SPLINE
SPL {X  -159.245, Y  +707.432, Z    +0.000, E1   -21.244, E3 +348737.690}
SPL {X  -162.277, Y  +686.791, Z    +0.000, E1   -10.607, E3 +348739.101}
SPL {X  -162.766, Y  +677.687, Z    +0.000, E1    -5.239, E3 +348741.291}
SPL {X  -162.820, Y  +671.059, Z    +0.000, E1    -0.934, E3 +348741.647}
SPL {X  -162.820, Y  +666.960, Z    +0.000, E1    +2.343, E3 +348741.923}
SPL {X  -162.820, Y  +662.610, Z    +0.000, E1    +6.209, E3 +348741.950}
SPL {X  -162.820, Y  +654.280, Z    +0.000, E1   +14.617, E3 +348742.282}
SPL {X  -162.820, Y  +638.947, Z    +0.000, E1   +31.033, E3 +348740.336}
SPL {X  -162.820, Y  +608.150, Z    +0.000, E1   +43.921, E3 +348766.569}
SPL {X  -162.820, Y  +574.255, Z    +0.000, E1   +46.562, E3 +348816.362}
ENDSPLINE

SPLINE
SPL {X  -162.820, Y  +579.440, Z    +0.000, E1   +42.450, E3 +348829.550}
ENDSPLINE

SPLINE
SPL {X  -162.820, Y  +573.350, Z    +0.000, E1   +42.340, E3 +348844.228}
SPL {X  -162.820, Y  +565.899, Z    +0.000, E1   +42.413, E3 +348860.811}
SPL {X  -162.820, Y  +560.278, Z    +0.000, E1   +42.308, E3 +348874.149}
SPL {X  -162.820, Y  +555.861, Z    +0.000, E1   +42.349, E3 +348883.997}
SPL {X  -162.820, Y  +550.633, Z    +0.000, E1   +42.421, E3 +348895.527}
SPL {X  -162.820, Y  +546.534, Z    +0.000, E1   +42.268, E3 +348905.736}
SPL {X  -162.820, Y  +539.632, Z    +0.000, E1   +42.488, E3 +348920.458}
SPL {X  -162.820, Y  +533.959, Z    +0.000, E1   +42.310, E3 +348934.154}
SPL {X  -162.820, Y  +527.661, Z    +0.000, E1   +42.425, E3 +348948.150}
SPL {X  -162.820, Y  +521.246, Z    +0.000, E1   +42.365, E3 +348962.903}
SPL {X  -162.820, Y  +515.708, Z    +0.000, E1   +42.333, E3 +348975.865}
SPL {X  -162.820, Y  +508.859, Z    +0.000, E1   +42.416, E3 +348991.007}
SPL {X  -162.820, Y  +501.651, Z    +0.000, E1   +42.423, E3 +349007.483}
SPL {X  -162.820, Y  +494.841, Z    +0.000, E1   +42.316, E3 +349023.593}
SPL {X  -162.820, Y  +489.758, Z    +0.000, E1   +42.464, E3 +349034.186}
SPL {X  -162.820, Y  +485.695, Z    +0.000, E1   +42.386, E3 +349044.022}
SPL {X  -162.820, Y  +464.528, Z    +0.000, E1   +47.611, E3 +349057.099}
SPL {X  -162.820, Y  +459.899, Z    +0.000, E1   +47.097, E3 +349068.942}
SPL {X  -162.820, Y  +455.990, Z    +0.000, E1   +46.212, E3 +349082.016}
SPL {X  -162.820, Y  +452.032, Z    +0.000, E1   +45.224, E3 +349095.801}
SPL {X  -162.820, Y  +446.617, Z    +0.000, E1   +44.768, E3 +349109.888}
SPL {X  -162.820, Y  +437.902, Z    +0.000, E1   +44.900, E3 +349127.464}
SPL {X  -162.820, Y  +429.336, Z    +0.000, E1   +44.917, E3 +349145.231}
SPL {X  -162.820, Y  +423.193, Z    +0.000, E1   +44.819, E3 +349158.490}
SPL {X  -162.820, Y  +416.810, Z    +0.000, E1   +44.932, E3 +349171.378}
SPL {X  -162.820, Y  +408.782, Z    +0.000, E1   +44.820, E3 +349188.809}
SPL {X  -162.820, Y  +401.619, Z    +0.000, E1   +44.978, E3 +349202.731}
SPL {X  -162.820, Y  +394.771, Z    +0.000, E1   +44.856, E3 +349217.970}
SPL {X  -162.820, Y  +387.883, Z    +0.000, E1   +44.837, E3 +349232.324}
SPL {X  -162.820, Y  +382.755, Z    +0.000, E1   +44.828, E3 +349243.117}
SPL {X  -162.796, Y  +377.700, Z    +0.000, E1   +44.829, E3 +349253.697}
SPL {X  -162.619, Y  +372.412, Z    +0.000, E1   +44.928, E3 +349264.156}
SPL {X  -162.311, Y  +367.633, Z    +0.000, E1   +44.798, E3 +349274.923}
SPL {X  -161.766, Y  +362.002, Z    +0.000, E1   +44.644, E3 +349287.682}
SPL {X  -161.043, Y  +356.508, Z    +0.000, E1   +44.528, E3 +349299.797}
SPL {X  -160.417, Y  +352.631, Z    +0.000, E1   +44.411, E3 +349308.528}
SPL {X  -159.536, Y  +347.962, Z    +0.000, E1   +44.302, E3 +349319.054}
SPL {X  -158.195, Y  +341.969, Z    +0.000, E1   +44.082, E3 +349332.837}
SPL {X  -156.950, Y  +337.174, Z    +0.000, E1   +43.768, E3 +349344.527}
SPL {X  -155.654, Y  +332.729, Z    +0.000, E1   +43.534, E3 +349355.169}
SPL {X  -154.189, Y  +328.191, Z    +0.000, E1   +43.338, E3 +349365.666}
SPL {X  -149.333, Y  +315.614, Z    +0.000, E1   +46.650, E3 +349372.982}
SPL {X  -142.680, Y  +302.060, Z    +0.000, E1   +42.084, E3 +349439.326}
ENDSPLINE

SPLINE
SPL {X  -151.184, Y  +320.053, Z    +0.000, E1   +32.435, E3 +349506.569}
SPL {X  -158.917, Y  +345.064, Z    +0.000, E1   +21.858, E3 +349507.917}
SPL {X  -161.350, Y  +358.672, Z    +0.000, E1   +15.089, E3 +349510.620}
SPL {X  -162.491, Y  +370.147, Z    +0.000, E1    +8.815, E3 +349513.555}
SPL {X  -162.771, Y  +376.522, Z    +0.000, E1    +5.005, E3 +349513.164}
SPL {X  -162.820, Y  +381.116, Z    +0.000, E1    +2.017, E3 +349513.498}
SPL {X  -162.820, Y  +384.427, Z    +0.000, E1    -0.390, E3 +349513.902}
SPL {X  -162.820, Y  +387.736, Z    +0.000, E1    -3.142, E3 +349513.183}
SPL {X  -162.820, Y  +391.456, Z    +0.000, E1    -6.603, E3 +349513.969}
SPL {X  -162.820, Y  +397.032, Z    +0.000, E1   -12.435, E3 +349513.416}
SPL {X  -162.820, Y  +406.111, Z    +0.000, E1   -22.010, E3 +349514.468}
SPL {X  -162.820, Y  +418.653, Z    +0.000, E1   -36.657, E3 +349508.821}
SPL {X  -162.820, Y  +440.590, Z    +0.000, E1   -50.152, E3 +349514.066}
SPL {X  -162.820, Y  +447.889, Z    +0.000, E1   -43.424, E3 +349545.212}
SPL {X  -162.820, Y  +478.087, Z    +0.000, E1   -45.903, E3 +349590.431}
ENDSPLINE

SPLINE
SPL {X  -162.820, Y  +474.900, Z    +0.000, E1   -42.394, E3 +349604.583}
ENDSPLINE

SPLINE
SPL {X  -162.820, Y  +480.895, Z    +0.000, E1   -42.223, E3 +349619.245}
SPL {X  -162.820, Y  +485.782, Z    +0.000, E1   -42.348, E3 +349629.590}
SPL {X  -162.820, Y  +489.480, Z    +0.000, E1   -42.230, E3 +349638.818}
SPL {X  -162.820, Y  +494.825, Z    +0.000, E1   -42.287, E3 +349650.765}
SPL {X  -162.820, Y  +501.023, Z    +0.000, E1   -42.347, E3 +349664.647}
SPL {X  -162.820, Y  +506.968, Z    +0.000, E1   -42.248, E3 +349678.838}
SPL {X  -162.820, Y  +513.215, Z    +0.000, E1   -42.304, E3 +349692.812}
SPL {X  -162.820, Y  +518.708, Z    +0.000, E1   -42.272, E3 +349705.534}
SPL {X  -162.820, Y  +525.147, Z    +0.000, E1   -42.298, E3 +349720.276}
SPL {X  -162.820, Y  +531.715, Z    +0.000, E1   -42.312, E3 +349735.102}
SPL {X  -162.820, Y  +537.459, Z    +0.000, E1   -42.308, E3 +349748.361}
SPL {X  -162.820, Y  +542.643, Z    +0.000, E1   -42.173, E3 +349760.953}
SPL {X  -162.820, Y  +549.160, Z    +0.000, E1   -42.387, E3 +349774.712}
SPL {X  -162.820, Y  +554.884, Z    +0.000, E1   -42.207, E3 +349788.798}
SPL {X  -162.820, Y  +561.114, Z    +0.000, E1   -42.336, E3 +349802.378}
SPL {X  -162.820, Y  +566.097, Z    +0.000, E1   -42.118, E3 +349814.988}
SPL {X  -162.820, Y  +571.654, Z    +0.000, E1   -42.313, E3 +349826.641}
SPL {X  -162.820, Y  +577.246, Z    +0.000, E1   -42.284, E3 +349839.607}
SPL {X  -162.820, Y  +582.233, Z    +0.000, E1   -42.188, E3 +349851.586}
SPL {X  -162.820, Y  +588.138, Z    +0.000, E1   -42.308, E3 +349864.484}
SPL {X  -162.820, Y  +593.999, Z    +0.000, E1   -42.301, E3 +349877.894}
SPL {X  -162.820, Y  +599.194, Z    +0.000, E1   -42.235, E3 +349890.199}
SPL {X  -162.820, Y  +604.595, Z    +0.000, E1   -42.290, E3 +349902.230}
SPL {X  -162.820, Y  +609.630, Z    +0.000, E1   -42.276, E3 +349913.856}
SPL {X  -162.820, Y  +614.392, Z    +0.000, E1   -42.242, E3 +349924.956}
SPL {X  -162.820, Y  +618.928, Z    +0.000, E1   -42.220, E3 +349935.482}
SPL {X  -162.820, Y  +625.176, Z    +0.000, E1   -42.323, E3 +349949.334}
SPL {X  -162.820, Y  +631.865, Z    +0.000, E1   -42.327, E3 +349964.547}
SPL {X  -162.820, Y  +637.189, Z    +0.000, E1   -42.236, E3 +349977.221}
SPL {X  -162.820, Y  +642.066, Z    +0.000, E1   -42.247, E3 +349988.344}
SPL {X  -162.820, Y  +646.907, Z    +0.000, E1   -42.249, E3 +349999.463}
SPL {X  -162.820, Y  +652.374, Z    +0.000, E1   -42.262, E3 +350011.901}
SPL {X  -162.820, Y  +657.439, Z    +0.000, E1   -42.251, E3 +350023.574}
SPL {X  -162.820, Y  +663.328, Z    +0.000, E1   -42.283, E3 +350036.976}
SPL {X  -162.820, Y  +669.078, Z    +0.000, E1   -42.263, E3 +350050.172}
SPL {X  -162.819, Y  +673.910, Z    +0.000, E1   -42.244, E3 +350061.366}
SPL {X  -162.670, Y  +680.491, Z    +0.000, E1   -42.282, E3 +350076.409}
SPL {X  -162.151, Y  +688.243, Z    +0.000, E1   -42.207, E3 +350094.610}
SPL {X  -161.446, Y  +694.609, Z    +0.000, E1   -42.094, E3 +350109.692}
SPL {X  -160.889, Y  +698.503, Z    +0.000, E1   -41.849, E3 +350119.966}
SPL {X  -160.100, Y  +703.138, Z    +0.000, E1   -41.824, E3 +350130.824}
SPL {X  -158.994, Y  +708.588, Z    +0.000, E1   -41.616, E3 +350144.544}
SPL {X  -157.709, Y  +713.973, Z    +0.000, E1   -41.360, E3 +350158.326}
SPL {X  -156.530, Y  +718.319, Z    +0.000, E1   -41.164, E3 +350169.271}
SPL {X  -155.547, Y  +721.618, Z    +0.000, E1   -40.968, E3 +350177.894}
SPL {X  -151.388, Y  +733.433, Z    +0.000, E1   -44.269, E3 +350185.597}
SPL {X  -144.352, Y  +748.818, Z    +0.000, E1   -40.701, E3 +350254.632}
SPL {X  -143.859, Y  +749.757, Z    +0.000, E1   -39.148, E3 +350282.580}
ENDSPLINE

SPLINE
SPL {X  -159.245, Y  +707.432, Z    +0.000, E1   -21.244, E3 +350314.614}
SPL {X  -162.277, Y  +686.791, Z    +0.000, E1   -10.607, E3 +350316.024}
SPL {X  -162.766, Y  +677.687, Z    +0.000, E1    -5.239, E3 +350318.214}
SPL {X  -162.820, Y  +671.059, Z    +0.000, E1    -0.934, E3 +350318.570}
SPL {X  -162.820, Y  +666.960, Z    +0.000, E1    +2.343, E3 +350318.846}
SPL {X  -162.820, Y  +662.610, Z    +0.000, E1    +6.209, E3 +350318.873}
SPL {X  -162.820, Y  +654.280, Z    +0.000, E1   +14.617, E3 +350319.206}
SPL {X  -162.820, Y  +638.947, Z    +0.000, E1   +31.033, E3 +350317.259}
SPL {X  -162.820, Y  +608.150, Z    +0.000, E1   +43.921, E3 +350343.492}
SPL {X  -162.820, Y  +574.255, Z    +0.000, E1   +46.562, E3 +350393.286}
ENDSPLINE

SPLINE
SPL {X  -162.820, Y  +579.440, Z    +0.000, E1   +42.450, E3 +350406.473}
ENDSPLINE

SPLINE
SPL {X  -162.820, Y  +574.443, Z    +0.000, E1   +42.333, E3 +350418.568}
SPL {X  -162.820, Y  +568.554, Z    +0.000, E1   +42.362, E3 +350431.930}
SPL {X  -162.820, Y  +563.699, Z    +0.000, E1   +42.375, E3 +350442.787}
SPL {X  -162.820, Y  +560.278, Z    +0.000, E1   +42.308, E3 +350451.072}
SPL {X  -162.820, Y  +554.421, Z    +0.000, E1   +42.414, E3 +350463.940}
SPL {X  -162.820, Y  +547.774, Z    +0.000, E1   +42.344, E3 +350479.513}
SPL {X  -162.820, Y  +541.056, Z    +0.000, E1   +42.452, E3 +350494.175}
SPL {X  -162.820, Y  +535.223, Z    +0.000, E1   +42.386, E3 +350507.868}
SPL {X  -162.820, Y  +529.084, Z    +0.000, E1   +42.400, E3 +350521.791}
SPL {X  -162.820, Y  +522.568, Z    +0.000, E1   +42.385, E3 +350536.821}
SPL {X  -162.820, Y  +515.708, Z    +0.000, E1   +42.333, E3 +350552.788}
SPL {X  -162.820, Y  +510.265, Z    +0.000, E1   +42.390, E3 +350564.750}
SPL {X  -162.820, Y  +505.746, Z    +0.000, E1   +42.400, E3 +350575.063}
SPL {X  -162.820, Y  +500.461, Z    +0.000, E1   +42.387, E3 +350587.190}
SPL {X  -162.820, Y  +494.841, Z    +0.000, E1   +42.316, E3 +350600.516}
SPL {X  -162.820, Y  +487.903, Z    +0.000, E1   +42.488, E3 +350615.339}
SPL {X  -162.820, Y  +484.250, Z    +0.000, E1   +42.201, E3 +350625.200}
SPL {X  -162.820, Y  +464.528, Z    +0.000, E1   +47.611, E3 +350634.022}
SPL {X  -162.820, Y  +459.899, Z    +0.000, E1   +47.097, E3 +350645.865}
SPL {X  -162.820, Y  +455.990, Z    +0.000, E1   +46.212, E3 +350658.939}
SPL {X  -162.820, Y  +452.032, Z    +0.000, E1   +45.224, E3 +350672.724}
SPL {X  -162.820, Y  +446.617, Z    +0.000, E1   +44.768, E3 +350686.811}
SPL {X  -162.820, Y  +437.902, Z    +0.000, E1   +44.900, E3 +350704.388}
SPL {X  -162.820, Y  +430.894, Z    +0.000, E1   +44.976, E3 +350718.373}
SPL {X  -162.820, Y  +425.053, Z    +0.000, E1   +44.824, E3 +350731.635}
SPL {X  -162.820, Y  +418.403, Z    +0.000, E1   +44.941, E3 +350744.748}
SPL {X  -162.820, Y  +412.479, Z    +0.000, E1   +44.780, E3 +350758.179}
SPL {X  -162.820, Y  +406.707, Z    +0.000, E1   +44.849, E3 +350769.751}
SPL {X  -162.820, Y  +400.166, Z    +0.000, E1   +44.948, E3 +350783.036}
SPL {X  -162.820, Y  +393.279, Z    +0.000, E1   +44.825, E3 +350798.038}
SPL {X  -162.820, Y  +387.883, Z    +0.000, E1   +44.837, E3 +350809.247}
SPL {X  -162.820, Y  +382.755, Z    +0.000, E1   +44.828, E3 +350820.040}
SPL {X  -162.796, Y  +377.700, Z    +0.000, E1   +44.829, E3 +350830.620}
SPL {X  -162.619, Y  +372.412, Z    +0.000, E1   +44.928, E3 +350841.079}
SPL {X  -162.311, Y  +367.633, Z    +0.000, E1   +44.798, E3 +350851.846}
SPL {X  -161.766, Y  +362.002, Z    +0.000, E1   +44.644, E3 +350864.605}
SPL {X  -161.043, Y  +356.508, Z    +0.000, E1   +44.528, E3 +350876.720}
SPL {X  -160.070, Y  +350.699, Z    +0.000, E1   +44.409, E3 +350889.672}
SPL {X  -158.853, Y  +344.776, Z    +0.000, E1   +44.148, E3 +350903.492}
SPL {X  -157.292, Y  +338.433, Z    +0.000, E1   +43.917, E3 +350918.170}
SPL {X  -155.654, Y  +332.729, Z    +0.000, E1   +43.534, E3 +350932.092}
SPL {X  -154.189, Y  +328.191, Z    +0.000, E1   +43.338, E3 +350942.589}
SPL {X  -149.333, Y  +315.614, Z    +0.000, E1   +46.650, E3 +350949.905}
SPL {X  -142.680, Y  +302.060, Z    +0.000, E1   +42.084, E3 +351016.249}
ENDSPLINE

SPLINE
SPL {X  -151.184, Y  +320.053, Z    +0.000, E1   +32.435, E3 +351083.492}
SPL {X  -158.917, Y  +345.064, Z    +0.000, E1   +21.858, E3 +351084.840}
SPL {X  -161.350, Y  +358.672, Z    +0.000, E1   +15.089, E3 +351087.543}
SPL {X  -162.491, Y  +370.147, Z    +0.000, E1    +8.815, E3 +351090.478}
SPL {X  -162.771, Y  +376.522, Z    +0.000, E1    +5.005, E3 +351090.087}
SPL {X  -162.820, Y  +383.029, Z    +0.000, E1    +0.769, E3 +351090.655}
SPL {X  -162.820, Y  +387.736, Z    +0.000, E1    -3.142, E3 +351090.106}
SPL {X  -162.820, Y  +392.770, Z    +0.000, E1    -7.830, E3 +351090.758}
SPL {X  -162.820, Y  +398.469, Z    +0.000, E1   -14.078, E3 +351090.210}
SPL {X  -162.820, Y  +406.111, Z    +0.000, E1   -22.010, E3 +351091.391}
SPL {X  -162.820, Y  +418.653, Z    +0.000, E1   -36.657, E3 +351085.744}
SPL {X  -162.820, Y  +440.590, Z    +0.000, E1   -50.152, E3 +351090.989}
SPL {X  -162.820, Y  +447.889, Z    +0.000, E1   -43.424, E3 +351122.135}
SPL {X  -162.820, Y  +479.020, Z    +0.000, E1   -47.189, E3 +351161.711}
ENDSPLINE

SPLINE
SPL {X  -162.820, Y  +474.886, Z    +0.000, E1   -43.721, E3 +351173.596}
ENDSPLINE

SPLINE
SPL {X  -162.820, Y  +477.319, Z    +0.000, E1   -42.306, E3 +351187.521}
SPL {X  -162.820, Y  +483.923, Z    +0.000, E1   -42.291, E3 +351202.728}
SPL {X  -162.820, Y  +489.480, Z    +0.000, E1   -42.230, E3 +351215.741}
SPL {X  -162.820, Y  +494.825, Z    +0.000, E1   -42.287, E3 +351227.688}
SPL {X  -162.820, Y  +501.023, Z    +0.000, E1   -42.347, E3 +351241.570}
SPL {X  -162.820, Y  +506.968, Z    +0.000, E1   -42.248, E3 +351255.761}
SPL {X  -162.820, Y  +513.215, Z    +0.000, E1   -42.304, E3 +351269.735}
SPL {X  -162.820, Y  +518.708, Z    +0.000, E1   -42.272, E3 +351282.457}
SPL {X  -162.820, Y  +525.147, Z    +0.000, E1   -42.298, E3 +351297.199}
SPL {X  -162.820, Y  +531.715, Z    +0.000, E1   -42.312, E3 +351312.025}
SPL {X  -162.820, Y  +537.459, Z    +0.000, E1   -42.308, E3 +351325.284}
SPL {X  -162.820, Y  +542.643, Z    +0.000, E1   -42.173, E3 +351337.876}
SPL {X  -162.820, Y  +549.160, Z    +0.000, E1   -42.387, E3 +351351.635}
SPL {X  -162.820, Y  +554.884, Z    +0.000, E1   -42.207, E3 +351365.721}
SPL {X  -162.820, Y  +561.114, Z    +0.000, E1   -42.336, E3 +351379.301}
SPL {X  -162.820, Y  +566.097, Z    +0.000, E1   -42.118, E3 +351391.911}
SPL {X  -162.820, Y  +571.654, Z    +0.000, E1   -42.313, E3 +351403.564}
SPL {X  -162.820, Y  +577.246, Z    +0.000, E1   -42.284, E3 +351416.530}
SPL {X  -162.820, Y  +582.233, Z    +0.000, E1   -42.188, E3 +351428.509}
SPL {X  -162.820, Y  +588.138, Z    +0.000, E1   -42.308, E3 +351441.407}
SPL {X  -162.820, Y  +593.999, Z    +0.000, E1   -42.301, E3 +351454.817}
SPL {X  -162.820, Y  +599.194, Z    +0.000, E1   -42.235, E3 +351467.122}
SPL {X  -162.820, Y  +604.595, Z    +0.000, E1   -42.290, E3 +351479.153}
SPL {X  -162.820, Y  +609.630, Z    +0.000, E1   -42.276, E3 +351490.779}
SPL {X  -162.820, Y  +614.392, Z    +0.000, E1   -42.242, E3 +351501.879}
SPL {X  -162.820, Y  +620.424, Z    +0.000, E1   -42.277, E3 +351515.627}
SPL {X  -162.820, Y  +626.430, Z    +0.000, E1   -42.291, E3 +351529.177}
SPL {X  -162.820, Y  +631.865, Z    +0.000, E1   -42.327, E3 +351541.470}
SPL {X  -162.820, Y  +637.189, Z    +0.000, E1   -42.236, E3 +351554.144}
SPL {X  -162.820, Y  +642.066, Z    +0.000, E1   -42.247, E3 +351565.267}
SPL {X  -162.820, Y  +646.907, Z    +0.000, E1   -42.249, E3 +351576.386}
SPL {X  -162.820, Y  +652.374, Z    +0.000, E1   -42.262, E3 +351588.824}
SPL {X  -162.820, Y  +657.439, Z    +0.000, E1   -42.251, E3 +351600.497}
SPL {X  -162.820, Y  +663.328, Z    +0.000, E1   -42.283, E3 +351613.899}
SPL {X  -162.820, Y  +669.078, Z    +0.000, E1   -42.263, E3 +351627.095}
SPL {X  -162.819, Y  +673.910, Z    +0.000, E1   -42.244, E3 +351638.289}
SPL {X  -162.729, Y  +678.944, Z    +0.000, E1   -42.273, E3 +351649.657}
SPL {X  -162.479, Y  +684.035, Z    +0.000, E1   -42.168, E3 +351661.994}
SPL {X  -162.026, Y  +689.560, Z    +0.000, E1   -42.192, E3 +351674.483}
SPL {X  -161.446, Y  +694.609, Z    +0.000, E1   -42.094, E3 +351686.615}
SPL {X  -160.681, Y  +699.806, Z    +0.000, E1   -41.866, E3 +351699.898}
SPL {X  -159.658, Y  +705.434, Z    +0.000, E1   -41.735, E3 +351713.528}
SPL {X  -158.727, Y  +709.780, Z    +0.000, E1   -41.560, E3 +351724.395}
SPL {X  -157.709, Y  +713.973, Z    +0.000, E1   -41.360, E3 +351735.249}
SPL {X  -156.530, Y  +718.319, Z    +0.000, E1   -41.164, E3 +351746.194}
SPL {X  -155.547, Y  +721.618, Z    +0.000, E1   -40.968, E3 +351754.818}
SPL {X  -151.388, Y  +733.433, Z    +0.000, E1   -44.269, E3 +351762.520}
SPL {X  -144.352, Y  +748.818, Z    +0.000, E1   -40.701, E3 +351831.555}
SPL {X  -143.859, Y  +749.757, Z    +0.000, E1   -39.148, E3 +351859.503}
ENDSPLINE

SPLINE
SPL {X  -159.245, Y  +707.432, Z    +0.000, E1   -21.244, E3 +351891.537}
SPL {X  -162.277, Y  +686.791, Z    +0.000, E1   -10.607, E3 +351892.947}
SPL {X  -162.766, Y  +677.687, Z    +0.000, E1    -5.239, E3 +351895.137}
SPL {X  -162.820, Y  +672.396, Z    +0.000, E1    -1.801, E3 +351895.925}
SPL {X  -162.820, Y  +667.851, Z    +0.000, E1    +1.551, E3 +351895.422}
SPL {X  -162.820, Y  +664.036, Z    +0.000, E1    +4.934, E3 +351896.141}
SPL {X  -162.820, Y  +661.024, Z    +0.000, E1    +7.880, E3 +351895.411}
SPL {X  -162.820, Y  +656.051, Z    +0.000, E1   +12.848, E3 +351896.278}
SPL {X  -162.820, Y  +650.794, Z    +0.000, E1   +18.580, E3 +351895.834}
SPL {X  -162.820, Y  +638.947, Z    +0.000, E1   +31.033, E3 +351894.182}
SPL {X  -162.820, Y  +608.150, Z    +0.000, E1   +43.921, E3 +351920.415}
SPL {X  -162.820, Y  +574.255, Z    +0.000, E1   +46.562, E3 +351970.209}
ENDSPLINE

SPLINE
SPL {X  -162.820, Y  +579.440, Z    +0.000, E1   +42.450, E3 +351983.396}
ENDSPLINE

SPLINE
SPL {X  -162.820, Y  +573.350, Z    +0.000, E1   +42.340, E3 +351998.074}
SPL {X  -162.820, Y  +565.899, Z    +0.000, E1   +42.413, E3 +352014.657}
SPL {X  -162.820, Y  +560.278, Z    +0.000, E1   +42.308, E3 +352027.995}
SPL {X  -162.820, Y  +554.421, Z    +0.000, E1   +42.414, E3 +352040.863}
SPL {X  -162.820, Y  +547.774, Z    +0.000, E1   +42.344, E3 +352056.436}
SPL {X  -162.820, Y  +541.056, Z    +0.000, E1   +42.452, E3 +352071.098}
SPL {X  -162.820, Y  +535.223, Z    +0.000, E1   +42.386, E3 +352084.791}
SPL {X  -162.820, Y  +529.084, Z    +0.000, E1   +42.400, E3 +352098.714}
SPL {X  -162.820, Y  +524.911, Z    +0.000, E1   +42.325, E3 +352108.560}
SPL {X  -162.820, Y  +519.984, Z    +0.000, E1   +42.385, E3 +352119.631}
SPL {X  -162.820, Y  +514.684, Z    +0.000, E1   +42.289, E3 +352132.202}
SPL {X  -162.820, Y  +508.859, Z    +0.000, E1   +42.416, E3 +352144.853}
SPL {X  -162.820, Y  +501.651, Z    +0.000, E1   +42.423, E3 +352161.329}
SPL {X  -162.820, Y  +496.578, Z    +0.000, E1   +42.329, E3 +352173.237}
SPL {X  -162.820, Y  +491.918, Z    +0.000, E1   +42.382, E3 +352183.731}
SPL {X  -162.820, Y  +485.695, Z    +0.000, E1   +42.386, E3 +352197.868}
SPL {X  -162.820, Y  +464.528, Z    +0.000, E1   +47.611, E3 +352210.946}
SPL {X  -162.820, Y  +459.899, Z    +0.000, E1   +47.097, E3 +352222.788}
SPL {X  -162.820, Y  +455.990, Z    +0.000, E1   +46.212, E3 +352235.862}
SPL {X  -162.820, Y  +452.032, Z    +0.000, E1   +45.224, E3 +352249.647}
SPL {X  -162.820, Y  +446.617, Z    +0.000, E1   +44.768, E3 +352263.734}
SPL {X  -162.820, Y  +437.902, Z    +0.000, E1   +44.900, E3 +352281.311}
SPL {X  -162.820, Y  +430.894, Z    +0.000, E1   +44.976, E3 +352295.296}
SPL {X  -162.820, Y  +425.053, Z    +0.000, E1   +44.824, E3 +352308.558}
SPL {X  -162.820, Y  +418.403, Z    +0.000, E1   +44.941, E3 +352321.671}
SPL {X  -162.820, Y  +412.479, Z    +0.000, E1   +44.780, E3 +352335.102}
SPL {X  -162.820, Y  +406.707, Z    +0.000, E1   +44.849, E3 +352346.674}
SPL {X  -162.820, Y  +401.619, Z    +0.000, E1   +44.978, E3 +352356.577}
SPL {X  -162.820, Y  +394.771, Z    +0.000, E1   +44.856, E3 +352371.816}
SPL {X  -162.820, Y  +387.883, Z    +0.000, E1   +44.837, E3 +352386.170}
SPL {X  -162.820, Y  +382.755, Z    +0.000, E1   +44.828, E3 +352396.963}
SPL {X  -162.796, Y  +377.700, Z    +0.000, E1   +44.829, E3 +352407.543}
SPL {X  -162.619, Y  +372.412, Z    +0.000, E1   +44.928, E3 +352418.002}
SPL {X  -162.311, Y  +367.633, Z    +0.000, E1   +44.798, E3 +352428.769}
SPL {X  -161.766, Y  +362.002, Z    +0.000, E1   +44.644, E3 +352441.528}
SPL {X  -161.043, Y  +356.508, Z    +0.000, E1   +44.528, E3 +352453.643}
SPL {X  -160.417, Y  +352.631, Z    +0.000, E1   +44.411, E3 +352462.374}
SPL {X  -159.536, Y  +347.962, Z    +0.000, E1   +44.302, E3 +352472.900}
SPL {X  -158.195, Y  +341.969, Z    +0.000, E1   +44.082, E3 +352486.683}
SPL {X  -156.950, Y  +337.174, Z    +0.000, E1   +43.768, E3 +352498.374}
SPL {X  -155.654, Y  +332.729, Z    +0.000, E1   +43.534, E3 +352509.015}
SPL {X  -153.067, Y  +324.996, Z    +0.000, E1   +44.257, E3 +352521.069}
SPL {X  -147.786, Y  +312.164, Z    +0.000, E1   +47.292, E3 +352529.800}
SPL {X  -142.680, Y  +302.060, Z    +0.000, E1   +42.084, E3 +352593.172}
ENDSPLINE

SPLINE
SPL {X  -151.184, Y  +320.053, Z    +0.000, E1   +32.435, E3 +352660.415}
SPL {X  -158.917, Y  +345.064, Z    +0.000, E1   +21.858, E3 +352661.763}
SPL {X  -161.350, Y  +358.672, Z    +0.000, E1   +15.089, E3 +352664.466}
SPL {X  -162.491, Y  +370.147, Z    +0.000, E1    +8.815, E3 +352667.401}
SPL {X  -162.816, Y  +379.394, Z    +0.000, E1    +3.267, E3 +352667.229}
SPL {X  -162.820, Y  +384.427, Z    +0.000, E1    -0.390, E3 +352667.748}
SPL {X  -162.820, Y  +387.736, Z    +0.000, E1    -3.142, E3 +352667.029}
SPL {X  -162.820, Y  +392.770, Z    +0.000, E1    -7.830, E3 +352667.681}
SPL {X  -162.820, Y  +398.469, Z    +0.000, E1   -14.078, E3 +352667.134}
SPL {X  -162.820, Y  +406.111, Z    +0.000, E1   -22.010, E3 +352668.314}
SPL {X  -162.820, Y  +418.653, Z    +0.000, E1   -36.657, E3 +352662.667}
SPL {X  -162.820, Y  +440.590, Z    +0.000, E1   -50.152, E3 +352667.912}
SPL {X  -162.820, Y  +447.889, Z    +0.000, E1   -43.424, E3 +352699.058}
SPL {X  -162.820, Y  +479.020, Z    +0.000, E1   -47.189, E3 +352738.634}
ENDSPLINE

SPLINE
SPL {X  -162.820, Y  +474.886, Z    +0.000, E1   -43.721, E3 +352750.519}
ENDSPLINE

SPLINE
SPL {X  -162.820, Y  +477.319, Z    +0.000, E1   -42.306, E3 +352764.444}
SPL {X  -162.820, Y  +483.923, Z    +0.000, E1   -42.291, E3 +352779.651}
SPL {X  -162.820, Y  +489.480, Z    +0.000, E1   -42.230, E3 +352792.664}
SPL {X  -162.820, Y  +494.825, Z    +0.000, E1   -42.287, E3 +352804.611}
SPL {X  -162.820, Y  +501.023, Z    +0.000, E1   -42.347, E3 +352818.493}
SPL {X  -162.820, Y  +506.968, Z    +0.000, E1   -42.248, E3 +352832.684}
SPL {X  -162.820, Y  +513.215, Z    +0.000, E1   -42.304, E3 +352846.658}
SPL {X  -162.820, Y  +518.708, Z    +0.000, E1   -42.272, E3 +352859.380}
SPL {X  -162.820, Y  +525.147, Z    +0.000, E1   -42.298, E3 +352874.122}
SPL {X  -162.820, Y  +531.715, Z    +0.000, E1   -42.312, E3 +352888.948}
SPL {X  -162.820, Y  +537.459, Z    +0.000, E1   -42.308, E3 +352902.207}
SPL {X  -162.820, Y  +542.643, Z    +0.000, E1   -42.173, E3 +352914.799}
SPL {X  -162.820, Y  +549.160, Z    +0.000, E1   -42.387, E3 +352928.558}
SPL {X  -162.820, Y  +554.884, Z    +0.000, E1   -42.207, E3 +352942.644}
SPL {X  -162.820, Y  +561.114, Z    +0.000, E1   -42.336, E3 +352956.224}
SPL {X  -162.820, Y  +566.097, Z    +0.000, E1   -42.118, E3 +352968.834}
SPL {X  -162.820, Y  +571.654, Z    +0.000, E1   -42.313, E3 +352980.487}
SPL {X  -162.820, Y  +577.246, Z    +0.000, E1   -42.284, E3 +352993.453}
SPL {X  -162.820, Y  +582.233, Z    +0.000, E1   -42.188, E3 +353005.432}
SPL {X  -162.820, Y  +588.138, Z    +0.000, E1   -42.308, E3 +353018.330}
SPL {X  -162.820, Y  +593.999, Z    +0.000, E1   -42.301, E3 +353031.740}
SPL {X  -162.820, Y  +599.194, Z    +0.000, E1   -42.235, E3 +353044.045}
SPL {X  -162.820, Y  +604.595, Z    +0.000, E1   -42.290, E3 +353056.076}
SPL {X  -162.820, Y  +609.630, Z    +0.000, E1   -42.276, E3 +353067.702}
SPL {X  -162.820, Y  +614.392, Z    +0.000, E1   -42.242, E3 +353078.802}
SPL {X  -162.820, Y  +620.424, Z    +0.000, E1   -42.277, E3 +353092.550}
SPL {X  -162.820, Y  +626.430, Z    +0.000, E1   -42.291, E3 +353106.100}
SPL {X  -162.820, Y  +631.865, Z    +0.000, E1   -42.327, E3 +353118.393}
SPL {X  -162.820, Y  +637.189, Z    +0.000, E1   -42.236, E3 +353131.067}
SPL {X  -162.820, Y  +642.066, Z    +0.000, E1   -42.247, E3 +353142.190}
SPL {X  -162.820, Y  +646.907, Z    +0.000, E1   -42.249, E3 +353153.309}
SPL {X  -162.820, Y  +652.374, Z    +0.000, E1   -42.262, E3 +353165.747}
SPL {X  -162.820, Y  +658.634, Z    +0.000, E1   -42.281, E3 +353180.104}
SPL {X  -162.820, Y  +664.480, Z    +0.000, E1   -42.257, E3 +353193.499}
SPL {X  -162.820, Y  +669.078, Z    +0.000, E1   -42.263, E3 +353204.018}
SPL {X  -162.819, Y  +673.910, Z    +0.000, E1   -42.244, E3 +353215.212}
SPL {X  -162.729, Y  +678.944, Z    +0.000, E1   -42.273, E3 +353226.580}
SPL {X  -162.479, Y  +684.035, Z    +0.000, E1   -42.168, E3 +353238.917}
SPL {X  -162.026, Y  +689.560, Z    +0.000, E1   -42.192, E3 +353251.406}
SPL {X  -161.446, Y  +694.609, Z    +0.000, E1   -42.094, E3 +353263.538}
SPL {X  -160.681, Y  +699.806, Z    +0.000, E1   -41.866, E3 +353276.821}
SPL {X  -159.658, Y  +705.434, Z    +0.000, E1   -41.735, E3 +353290.451}
SPL {X  -158.502, Y  +710.748, Z    +0.000, E1   -41.532, E3 +353303.798}
SPL {X  -157.452, Y  +714.962, Z    +0.000, E1   -41.276, E3 +353314.794}
SPL {X  -156.530, Y  +718.319, Z    +0.000, E1   -41.164, E3 +353323.117}
SPL {X  -155.547, Y  +721.618, Z    +0.000, E1   -40.968, E3 +353331.741}
SPL {X  -151.388, Y  +733.433, Z    +0.000, E1   -44.269, E3 +353339.443}
SPL {X  -144.352, Y  +748.818, Z    +0.000, E1   -40.701, E3 +353408.478}
SPL {X  -143.859, Y  +749.757, Z    +0.000, E1   -39.148, E3 +353436.426}
ENDSPLINE

SPLINE
SPL {X  -159.245, Y  +707.432, Z    +0.000, E1   -21.244, E3 +353468.460}
SPL {X  -162.277, Y  +686.791, Z    +0.000, E1   -10.607, E3 +353469.870}
SPL {X  -162.766, Y  +677.687, Z    +0.000, E1    -5.239, E3 +353472.060}
SPL {X  -162.820, Y  +671.059, Z    +0.000, E1    -0.934, E3 +353472.416}
SPL {X  -162.820, Y  +666.960, Z    +0.000, E1    +2.343, E3 +353472.692}
SPL {X  -162.820, Y  +662.610, Z    +0.000, E1    +6.209, E3 +353472.719}
SPL {X  -162.820, Y  +654.280, Z    +0.000, E1   +14.617, E3 +353473.052}
SPL {X  -162.820, Y  +638.947, Z    +0.000, E1   +31.033, E3 +353471.105}
SPL {X  -162.820, Y  +608.150, Z    +0.000, E1   +43.921, E3 +353497.338}
SPL {X  -162.820, Y  +574.255, Z    +0.000, E1   +46.562, E3 +353547.132}
ENDSPLINE

SPLINE
SPL {X  -162.820, Y  +579.440, Z    +0.000, E1   +42.450, E3 +353560.319}
ENDSPLINE

SPLINE
SPL {X  -162.820, Y  +574.443, Z    +0.000, E1   +42.333, E3 +353572.414}
SPL {X  -162.820, Y  +568.554, Z    +0.000, E1   +42.362, E3 +353585.776}
SPL {X  -162.820, Y  +561.474, Z    +0.000, E1   +42.369, E3 +353601.961}
SPL {X  -162.820, Y  +554.421, Z    +0.000, E1   +42.414, E3 +353617.786}
SPL {X  -162.820, Y  +547.774, Z    +0.000, E1   +42.344, E3 +353633.359}
SPL {X  -162.820, Y  +541.056, Z    +0.000, E1   +42.452, E3 +353648.021}
SPL {X  -162.820, Y  +535.223, Z    +0.000, E1   +42.386, E3 +353661.714}
SPL {X  -162.820, Y  +529.084, Z    +0.000, E1   +42.400, E3 +353675.637}
SPL {X  -162.820, Y  +522.568, Z    +0.000, E1   +42.385, E3 +353690.667}
SPL {X  -162.820, Y  +515.708, Z    +0.000, E1   +42.333, E3 +353706.634}
SPL {X  -162.820, Y  +508.859, Z    +0.000, E1   +42.416, E3 +353721.776}
SPL {X  -162.820, Y  +501.651, Z    +0.000, E1   +42.423, E3 +353738.252}
SPL {X  -162.820, Y  +494.841, Z    +0.000, E1   +42.316, E3 +353754.362}
SPL {X  -162.820, Y  +486.958, Z    +0.000, E1   +42.460, E3 +353771.655}
SPL {X  -162.820, Y  +466.305, Z    +0.000, E1   +47.564, E3 +353784.662}
SPL {X  -162.820, Y  +460.790, Z    +0.000, E1   +47.323, E3 +353796.838}
SPL {X  -162.820, Y  +455.990, Z    +0.000, E1   +46.212, E3 +353812.785}
SPL {X  -162.820, Y  +452.032, Z    +0.000, E1   +45.224, E3 +353826.570}
SPL {X  -162.820, Y  +446.617, Z    +0.000, E1   +44.768, E3 +353840.657}
SPL {X  -162.820, Y  +437.902, Z    +0.000, E1   +44.900, E3 +353858.234}
SPL {X  -162.820, Y  +430.894, Z    +0.000, E1   +44.976, E3 +353872.219}
SPL {X  -162.820, Y  +425.053, Z    +0.000, E1   +44.824, E3 +353885.481}
SPL {X  -162.820, Y  +416.810, Z    +0.000, E1   +44.932, E3 +353902.148}
SPL {X  -162.820, Y  +408.782, Z    +0.000, E1   +44.820, E3 +353919.578}
SPL {X  -162.820, Y  +401.619, Z    +0.000, E1   +44.978, E3 +353933.500}
SPL {X  -162.820, Y  +394.771, Z    +0.000, E1   +44.856, E3 +353948.739}
SPL {X  -162.820, Y  +387.883, Z    +0.000, E1   +44.837, E3 +353963.093}
SPL {X  -162.820, Y  +382.755, Z    +0.000, E1   +44.828, E3 +353973.886}
SPL {X  -162.796, Y  +377.700, Z    +0.000, E1   +44.829, E3 +353984.466}
SPL {X  -162.619, Y  +372.412, Z    +0.000, E1   +44.928, E3 +353994.925}
SPL {X  -162.311, Y  +367.633, Z    +0.000, E1   +44.798, E3 +354005.693}
SPL {X  -161.766, Y  +362.002, Z    +0.000, E1   +44.644, E3 +354018.451}
SPL {X  -161.043, Y  +356.508, Z    +0.000, E1   +44.528, E3 +354030.566}
SPL {X  -160.070, Y  +350.699, Z    +0.000, E1   +44.409, E3 +354043.518}
SPL {X  -158.853, Y  +344.776, Z    +0.000, E1   +44.148, E3 +354057.338}
SPL {X  -157.292, Y  +338.433, Z    +0.000, E1   +43.917, E3 +354072.017}
SPL {X  -155.654, Y  +332.729, Z    +0.000, E1   +43.534, E3 +354085.938}
SPL {X  -154.189, Y  +328.191, Z    +0.000, E1   +43.338, E3 +354096.435}
SPL {X  -149.333, Y  +315.614, Z    +0.000, E1   +46.650, E3 +354103.751}
SPL {X  -142.680, Y  +302.060, Z    +0.000, E1   +42.084, E3 +354170.095}
ENDSPLINE

SPLINE
SPL {X  -151.184, Y  +320.053, Z    +0.000, E1   +32.435, E3 +354237.338}
SPL {X  -158.917, Y  +345.064, Z    +0.000, E1   +21.858, E3 +354238.687}
SPL {X  -161.350, Y  +358.672, Z    +0.000, E1   +15.089, E3 +354241.389}
SPL {X  -162.491, Y  +370.147, Z    +0.000, E1    +8.815, E3 +354244.324}
SPL {X  -162.771, Y  +376.522, Z    +0.000, E1    +5.005, E3 +354243.933}
SPL {X  -162.820, Y  +383.029, Z    +0.000, E1    +0.769, E3 +354244.501}
SPL {X  -162.820, Y  +387.736, Z    +0.000, E1    -3.142, E3 +354243.952}
SPL {X  -162.820, Y  +392.770, Z    +0.000, E1    -7.830, E3 +354244.604}
SPL {X  -162.820, Y  +398.469, Z    +0.000, E1   -14.078, E3 +354244.057}
SPL {X  -162.820, Y  +406.111, Z    +0.000, E1   -22.010, E3 +354245.237}
SPL {X  -162.820, Y  +418.653, Z    +0.000, E1   -36.657, E3 +354239.590}
SPL {X  -162.820, Y  +440.590, Z    +0.000, E1   -50.152, E3 +354244.835}
SPL {X  -162.820, Y  +447.889, Z    +0.000, E1   -43.424, E3 +354275.981}
SPL {X  -162.820, Y  +478.087, Z    +0.000, E1   -45.903, E3 +354321.200}
ENDSPLINE

SPLINE
SPL {X  -162.820, Y  +474.900, Z    +0.000, E1   -42.394, E3 +354335.353}
ENDSPLINE

SPLINE
SPL {X  -162.820, Y  +480.895, Z    +0.000, E1   -42.223, E3 +354350.014}
SPL {X  -162.820, Y  +485.782, Z    +0.000, E1   -42.348, E3 +354360.360}
SPL {X  -162.820, Y  +489.480, Z    +0.000, E1   -42.230, E3 +354369.587}
SPL {X  -162.820, Y  +494.825, Z    +0.000, E1   -42.287, E3 +354381.534}
SPL {X  -162.820, Y  +501.023, Z    +0.000, E1   -42.347, E3 +354395.416}
SPL {X  -162.820, Y  +506.968, Z    +0.000, E1   -42.248, E3 +354409.607}
SPL {X  -162.820, Y  +513.215, Z    +0.000, E1   -42.304, E3 +354423.582}
SPL {X  -162.820, Y  +518.708, Z    +0.000, E1   -42.272, E3 +354436.303}
SPL {X  -162.820, Y  +525.147, Z    +0.000, E1   -42.298, E3 +354451.045}
SPL {X  -162.820, Y  +531.715, Z    +0.000, E1   -42.312, E3 +354465.871}
SPL {X  -162.820, Y  +537.459, Z    +0.000, E1   -42.308, E3 +354479.130}
SPL {X  -162.820, Y  +542.643, Z    +0.000, E1   -42.173, E3 +354491.723}
SPL {X  -162.820, Y  +549.160, Z    +0.000, E1   -42.387, E3 +354505.481}
SPL {X  -162.820, Y  +554.884, Z    +0.000, E1   -42.207, E3 +354519.567}
SPL {X  -162.820, Y  +561.114, Z    +0.000, E1   -42.336, E3 +354533.147}
SPL {X  -162.820, Y  +566.097, Z    +0.000, E1   -42.118, E3 +354545.757}
SPL {X  -162.820, Y  +571.654, Z    +0.000, E1   -42.313, E3 +354557.410}
SPL {X  -162.820, Y  +577.246, Z    +0.000, E1   -42.284, E3 +354570.376}
SPL {X  -162.820, Y  +582.233, Z    +0.000, E1   -42.188, E3 +354582.355}
SPL {X  -162.820, Y  +588.138, Z    +0.000, E1   -42.308, E3 +354595.253}
SPL {X  -162.820, Y  +593.999, Z    +0.000, E1   -42.301, E3 +354608.663}
SPL {X  -162.820, Y  +599.194, Z    +0.000, E1   -42.235, E3 +354620.968}
SPL {X  -162.820, Y  +604.595, Z    +0.000, E1   -42.290, E3 +354633.000}
SPL {X  -162.820, Y  +609.630, Z    +0.000, E1   -42.276, E3 +354644.625}
SPL {X  -162.820, Y  +614.392, Z    +0.000, E1   -42.242, E3 +354655.726}
SPL {X  -162.820, Y  +620.424, Z    +0.000, E1   -42.277, E3 +354669.473}
SPL {X  -162.820, Y  +626.430, Z    +0.000, E1   -42.291, E3 +354683.023}
SPL {X  -162.820, Y  +631.865, Z    +0.000, E1   -42.327, E3 +354695.317}
SPL {X  -162.820, Y  +637.189, Z    +0.000, E1   -42.236, E3 +354707.991}
SPL {X  -162.820, Y  +642.066, Z    +0.000, E1   -42.247, E3 +354719.113}
SPL {X  -162.820, Y  +646.907, Z    +0.000, E1   -42.249, E3 +354730.232}
SPL {X  -162.820, Y  +652.374, Z    +0.000, E1   -42.262, E3 +354742.670}
SPL {X  -162.820, Y  +657.439, Z    +0.000, E1   -42.251, E3 +354754.343}
SPL {X  -162.820, Y  +663.328, Z    +0.000, E1   -42.283, E3 +354767.745}
SPL {X  -162.820, Y  +669.078, Z    +0.000, E1   -42.263, E3 +354780.941}
SPL {X  -162.819, Y  +673.910, Z    +0.000, E1   -42.244, E3 +354792.136}
SPL {X  -162.729, Y  +678.944, Z    +0.000, E1   -42.273, E3 +354803.503}
SPL {X  -162.479, Y  +684.035, Z    +0.000, E1   -42.168, E3 +354815.841}
SPL {X  -162.026, Y  +689.560, Z    +0.000, E1   -42.192, E3 +354828.329}
SPL {X  -161.446, Y  +694.609, Z    +0.000, E1   -42.094, E3 +354840.461}
SPL {X  -160.889, Y  +698.503, Z    +0.000, E1   -41.849, E3 +354850.735}
SPL {X  -160.100, Y  +703.138, Z    +0.000, E1   -41.824, E3 +354861.594}
SPL {X  -158.994, Y  +708.588, Z    +0.000, E1   -41.616, E3 +354875.313}
SPL {X  -157.709, Y  +713.973, Z    +0.000, E1   -41.360, E3 +354889.095}
SPL {X  -156.530, Y  +718.319, Z    +0.000, E1   -41.164, E3 +354900.040}
SPL {X  -155.547, Y  +721.618, Z    +0.000, E1   -40.968, E3 +354908.664}
SPL {X  -151.388, Y  +733.433, Z    +0.000, E1   -44.269, E3 +354916.366}
SPL {X  -144.352, Y  +748.818, Z    +0.000, E1   -40.701, E3 +354985.401}
SPL {X  -143.859, Y  +749.757, Z    +0.000, E1   -39.148, E3 +355013.350}
ENDSPLINE

SPLINE
SPL {X  -159.245, Y  +707.432, Z    +0.000, E1   -21.244, E3 +355045.383}
SPL {X  -162.277, Y  +686.791, Z    +0.000, E1   -10.607, E3 +355046.793}
SPL {X  -162.766, Y  +677.687, Z    +0.000, E1    -5.239, E3 +355048.983}
SPL {X  -162.820, Y  +671.059, Z    +0.000, E1    -0.934, E3 +355049.339}
SPL {X  -162.820, Y  +665.599, Z    +0.000, E1    +3.424, E3 +355049.789}
SPL {X  -162.820, Y  +661.024, Z    +0.000, E1    +7.880, E3 +355049.257}
SPL {X  -162.820, Y  +654.280, Z    +0.000, E1   +14.617, E3 +355049.975}
SPL {X  -162.820, Y  +638.947, Z    +0.000, E1   +31.033, E3 +355048.028}
SPL {X  -162.820, Y  +608.150, Z    +0.000, E1   +43.921, E3 +355074.261}
SPL {X  -162.820, Y  +574.255, Z    +0.000, E1   +46.562, E3 +355124.055}
ENDSPLINE

SPLINE
SPL {X  -162.820, Y  +579.440, Z    +0.000, E1   +42.450, E3 +355137.242}
ENDSPLINE

SPLINE
SPL {X  -162.820, Y  +574.443, Z    +0.000, E1   +42.333, E3 +355149.337}
SPL {X  -162.820, Y  +568.554, Z    +0.000, E1   +42.362, E3 +355162.699}
SPL {X  -162.820, Y  +561.474, Z    +0.000, E1   +42.369, E3 +355178.885}
SPL {X  -162.820, Y  +554.421, Z    +0.000, E1   +42.414, E3 +355194.709}
SPL {X  -162.820, Y  +547.774, Z    +0.000, E1   +42.344, E3 +355210.282}
SPL {X  -162.820, Y  +541.056, Z    +0.000, E1   +42.452, E3 +355224.944}
SPL {X  -162.820, Y  +535.223, Z    +0.000, E1   +42.386, E3 +355238.637}
SPL {X  -162.820, Y  +529.084, Z    +0.000, E1   +42.400, E3 +355252.560}
SPL {X  -162.820, Y  +524.911, Z    +0.000, E1   +42.325, E3 +355262.406}
SPL {X  -162.820, Y  +519.984, Z    +0.000, E1   +42.385, E3 +355273.477}
SPL {X  -162.820, Y  +512.536, Z    +0.000, E1   +42.385, E3 +355290.587}
SPL {X  -162.820, Y  +505.746, Z    +0.000, E1   +42.400, E3 +355305.832}
SPL {X  -162.820, Y  +500.461, Z    +0.000, E1   +42.387, E3 +355317.959}
SPL {X  -162.820, Y  +494.841, Z    +0.000, E1   +42.316, E3 +355331.285}
SPL {X  -162.820, Y  +486.958, Z    +0.000, E1   +42.460, E3 +355348.578}
SPL {X  -162.820, Y  +466.305, Z    +0.000, E1   +47.564, E3 +355361.585}
SPL {X  -162.820, Y  +462.532, Z    +0.000, E1   +47.610, E3 +355368.469}
SPL {X  -162.820, Y  +458.830, Z    +0.000, E1   +46.994, E3 +355379.470}
SPL {X  -162.820, Y  +455.537, Z    +0.000, E1   +45.900, E3 +355392.289}
SPL {X  -162.820, Y  +451.000, Z    +0.000, E1   +45.084, E3 +355406.664}
SPL {X  -162.820, Y  +442.850, Z    +0.000, E1   +44.856, E3 +355425.040}
SPL {X  -162.820, Y  +435.902, Z    +0.000, E1   +44.853, E3 +355439.405}
SPL {X  -162.820, Y  +429.336, Z    +0.000, E1   +44.917, E3 +355452.924}
SPL {X  -162.820, Y  +423.193, Z    +0.000, E1   +44.819, E3 +355466.183}
SPL {X  -162.820, Y  +416.810, Z    +0.000, E1   +44.932, E3 +355479.071}
SPL {X  -162.820, Y  +408.782, Z    +0.000, E1   +44.820, E3 +355496.501}
SPL {X  -162.820, Y  +401.619, Z    +0.000, E1   +44.978, E3 +355510.423}
SPL {X  -162.820, Y  +394.771, Z    +0.000, E1   +44.856, E3 +355525.662}
SPL {X  -162.820, Y  +387.883, Z    +0.000, E1   +44.837, E3 +355540.016}
SPL {X  -162.820, Y  +382.755, Z    +0.000, E1   +44.828, E3 +355550.809}
SPL {X  -162.796, Y  +377.700, Z    +0.000, E1   +44.829, E3 +355561.389}
SPL {X  -162.619, Y  +372.412, Z    +0.000, E1   +44.928, E3 +355571.849}
SPL {X  -162.311, Y  +367.633, Z    +0.000, E1   +44.798, E3 +355582.616}
SPL {X  -161.766, Y  +362.002, Z    +0.000, E1   +44.644, E3 +355595.374}
SPL {X  -161.043, Y  +356.508, Z    +0.000, E1   +44.528, E3 +355607.489}
SPL {X  -160.417, Y  +352.631, Z    +0.000, E1   +44.411, E3 +355616.220}
SPL {X  -159.536, Y  +347.962, Z    +0.000, E1   +44.302, E3 +355626.747}
SPL {X  -158.195, Y  +341.969, Z    +0.000, E1   +44.082, E3 +355640.529}
SPL {X  -156.950, Y  +337.174, Z    +0.000, E1   +43.768, E3 +355652.220}
SPL {X  -155.654, Y  +332.729, Z    +0.000, E1   +43.534, E3 +355662.862}
SPL {X  -153.067, Y  +324.996, Z    +0.000, E1   +44.257, E3 +355674.916}
SPL {X  -147.786, Y  +312.164, Z    +0.000, E1   +47.292, E3 +355683.646}
SPL {X  -142.680, Y  +302.060, Z    +0.000, E1   +42.084, E3 +355747.018}
ENDSPLINE

SPLINE
SPL {X  -151.184, Y  +320.053, Z    +0.000, E1   +32.435, E3 +355814.261}
SPL {X  -158.917, Y  +345.064, Z    +0.000, E1   +21.858, E3 +355815.610}
SPL {X  -161.350, Y  +358.672, Z    +0.000, E1   +15.089, E3 +355818.312}
SPL {X  -162.491, Y  +370.147, Z    +0.000, E1    +8.815, E3 +355821.247}
SPL {X  -162.771, Y  +376.522, Z    +0.000, E1    +5.005, E3 +355820.856}
SPL {X  -162.820, Y  +381.116, Z    +0.000, E1    +2.017, E3 +355821.190}
SPL {X  -162.820, Y  +384.427, Z    +0.000, E1    -0.390, E3 +355821.595}
SPL {X  -162.820, Y  +387.736, Z    +0.000, E1    -3.142, E3 +355820.875}
SPL {X  -162.820, Y  +391.456, Z    +0.000, E1    -6.603, E3 +355821.662}
SPL {X  -162.820, Y  +397.032, Z    +0.000, E1   -12.435, E3 +355821.109}
SPL {X  -162.820, Y  +406.111, Z    +0.000, E1   -22.010, E3 +355822.160}
SPL {X  -162.820, Y  +418.653, Z    +0.000, E1   -36.657, E3 +355816.513}
SPL {X  -162.820, Y  +440.590, Z    +0.000, E1   -50.152, E3 +355821.758}
SPL {X  -162.820, Y  +447.889, Z    +0.000, E1   -43.424, E3 +355852.904}
SPL {X  -162.820, Y  +479.020, Z    +0.000, E1   -47.189, E3 +355892.480}
ENDSPLINE

SPLINE
SPL {X  -162.820, Y  +474.886, Z    +0.000, E1   -43.721, E3 +355904.365}
ENDSPLINE

SPLINE
SPL {X  -162.820, Y  +476.137, Z    +0.000, E1   -42.304, E3 +355915.478}
SPL {X  -162.820, Y  +480.895, Z    +0.000, E1   -42.223, E3 +355926.937}
SPL {X  -162.820, Y  +485.782, Z    +0.000, E1   -42.348, E3 +355937.283}
SPL {X  -162.820, Y  +489.480, Z    +0.000, E1   -42.230, E3 +355946.510}
SPL {X  -162.820, Y  +494.825, Z    +0.000, E1   -42.287, E3 +355958.457}
SPL {X  -162.820, Y  +501.909, Z    +0.000, E1   -42.324, E3 +355974.644}
SPL {X  -162.820, Y  +508.157, Z    +0.000, E1   -42.280, E3 +355988.974}
SPL {X  -162.820, Y  +513.215, Z    +0.000, E1   -42.304, E3 +356000.505}
SPL {X  -162.820, Y  +520.311, Z    +0.000, E1   -42.317, E3 +356016.803}
SPL {X  -162.820, Y  +526.529, Z    +0.000, E1   -42.247, E3 +356031.272}
SPL {X  -162.820, Y  +531.715, Z    +0.000, E1   -42.312, E3 +356042.794}
SPL {X  -162.820, Y  +537.459, Z    +0.000, E1   -42.308, E3 +356056.053}
SPL {X  -162.820, Y  +542.643, Z    +0.000, E1   -42.173, E3 +356068.646}
SPL {X  -162.820, Y  +549.160, Z    +0.000, E1   -42.387, E3 +356082.404}
SPL {X  -162.820, Y  +554.884, Z    +0.000, E1   -42.207, E3 +356096.490}
SPL {X  -162.820, Y  +561.114, Z    +0.000, E1   -42.336, E3 +356110.070}
SPL {X  -162.820, Y  +566.097, Z    +0.000, E1   -42.118, E3 +356122.680}
SPL {X  -162.820, Y  +571.654, Z    +0.000, E1   -42.313, E3 +356134.333}
SPL {X  -162.820, Y  +577.246, Z    +0.000, E1   -42.284, E3 +356147.299}
SPL {X  -162.820, Y  +582.233, Z    +0.000, E1   -42.188, E3 +356159.278}
SPL {X  -162.820, Y  +588.138, Z    +0.000, E1   -42.308, E3 +356172.176}
SPL {X  -162.820, Y  +593.999, Z    +0.000, E1   -42.301, E3 +356185.587}
SPL {X  -162.820, Y  +599.194, Z    +0.000, E1   -42.235, E3 +356197.891}
SPL {X  -162.820, Y  +604.595, Z    +0.000, E1   -42.290, E3 +356209.923}
SPL {X  -162.820, Y  +609.630, Z    +0.000, E1   -42.276, E3 +356221.549}
SPL {X  -162.820, Y  +614.392, Z    +0.000, E1   -42.242, E3 +356232.649}
SPL {X  -162.820, Y  +620.424, Z    +0.000, E1   -42.277, E3 +356246.396}
SPL {X  -162.820, Y  +626.430, Z    +0.000, E1   -42.291, E3 +356259.946}
SPL {X  -162.820, Y  +631.865, Z    +0.000, E1   -42.327, E3 +356272.240}
SPL {X  -162.820, Y  +637.189, Z    +0.000, E1   -42.236, E3 +356284.914}
SPL {X  -162.820, Y  +642.066, Z    +0.000, E1   -42.247, E3 +356296.036}
SPL {X  -162.820, Y  +646.907, Z    +0.000, E1   -42.249, E3 +356307.155}
SPL {X  -162.820, Y  +652.374, Z    +0.000, E1   -42.262, E3 +356319.593}
SPL {X  -162.820, Y  +657.439, Z    +0.000, E1   -42.251, E3 +356331.266}
SPL {X  -162.820, Y  +663.328, Z    +0.000, E1   -42.283, E3 +356344.668}
SPL {X  -162.820, Y  +669.078, Z    +0.000, E1   -42.263, E3 +356357.864}
SPL {X  -162.819, Y  +673.910, Z    +0.000, E1   -42.244, E3 +356369.059}
SPL {X  -162.729, Y  +678.944, Z    +0.000, E1   -42.273, E3 +356380.426}
SPL {X  -162.479, Y  +684.035, Z    +0.000, E1   -42.168, E3 +356392.764}
SPL {X  -162.026, Y  +689.560, Z    +0.000, E1   -42.192, E3 +356405.252}
SPL {X  -161.446, Y  +694.609, Z    +0.000, E1   -42.094, E3 +356417.384}
SPL {X  -160.681, Y  +699.806, Z    +0.000, E1   -41.866, E3 +356430.667}
SPL {X  -159.658, Y  +705.434, Z    +0.000, E1   -41.735, E3 +356444.297}
SPL {X  -158.502, Y  +710.748, Z    +0.000, E1   -41.532, E3 +356457.645}
SPL {X  -157.452, Y  +714.962, Z    +0.000, E1   -41.276, E3 +356468.640}
SPL {X  -156.530, Y  +718.319, Z    +0.000, E1   -41.164, E3 +356476.963}
SPL {X  -155.547, Y  +721.618, Z    +0.000, E1   -40.968, E3 +356485.587}
SPL {X  -151.388, Y  +733.433, Z    +0.000, E1   -44.269, E3 +356493.290}
SPL {X  -144.352, Y  +748.818, Z    +0.000, E1   -40.701, E3 +356562.324}
SPL {X  -143.859, Y  +749.757, Z    +0.000, E1   -39.148, E3 +356590.273}
ENDSPLINE

SPLINE
SPL {X  -159.245, Y  +707.432, Z    +0.000, E1   -21.244, E3 +356622.306}
SPL {X  -162.277, Y  +686.791, Z    +0.000, E1   -10.607, E3 +356623.716}
SPL {X  -162.766, Y  +677.687, Z    +0.000, E1    -5.239, E3 +356625.906}
SPL {X  -162.820, Y  +671.059, Z    +0.000, E1    -0.934, E3 +356626.262}
SPL {X  -162.820, Y  +665.599, Z    +0.000, E1    +3.424, E3 +356626.712}
SPL {X  -162.820, Y  +661.024, Z    +0.000, E1    +7.880, E3 +356626.180}
SPL {X  -162.820, Y  +656.051, Z    +0.000, E1   +12.848, E3 +356627.047}
SPL {X  -162.820, Y  +650.794, Z    +0.000, E1   +18.580, E3 +356626.603}
SPL {X  -162.820, Y  +638.947, Z    +0.000, E1   +31.033, E3 +356624.951}
SPL {X  -162.820, Y  +608.150, Z    +0.000, E1   +43.921, E3 +356651.184}
SPL {X  -162.820, Y  +574.255, Z    +0.000, E1   +46.562, E3 +356700.978}
ENDSPLINE

SPLINE
SPL {X  -162.820, Y  +579.440, Z    +0.000, E1   +42.450, E3 +356714.165}
ENDSPLINE

SPLINE
SPL {X  -162.820, Y  +574.443, Z    +0.000, E1   +42.333, E3 +356726.260}
SPL {X  -162.820, Y  +568.554, Z    +0.000, E1   +42.362, E3 +356739.622}
SPL {X  -162.820, Y  +561.474, Z    +0.000, E1   +42.369, E3 +356755.808}
SPL {X  -162.820, Y  +555.861, Z    +0.000, E1   +42.349, E3 +356768.612}
SPL {X  -162.820, Y  +550.633, Z    +0.000, E1   +42.421, E3 +356780.142}
SPL {X  -162.820, Y  +546.534, Z    +0.000, E1   +42.268, E3 +356790.352}
SPL {X  -162.820, Y  +539.632, Z    +0.000, E1   +42.488, E3 +356805.073}
SPL {X  -162.820, Y  +533.959, Z    +0.000, E1   +42.310, E3 +356818.770}
SPL {X  -162.820, Y  +527.661, Z    +0.000, E1   +42.425, E3 +356832.765}
SPL {X  -162.820, Y  +521.246, Z    +0.000, E1   +42.365, E3 +356847.518}
SPL {X  -162.820, Y  +515.708, Z    +0.000, E1   +42.333, E3 +356860.481}
SPL {X  -162.820, Y  +510.265, Z    +0.000, E1   +42.390, E3 +356872.442}
SPL {X  -162.820, Y  +505.746, Z    +0.000, E1   +42.400, E3 +356882.755}
SPL {X  -162.820, Y  +500.461, Z    +0.000, E1   +42.387, E3 +356894.882}
SPL {X  -162.820, Y  +494.841, Z    +0.000, E1   +42.316, E3 +356908.208}
SPL {X  -162.820, Y  +486.958, Z    +0.000, E1   +42.460, E3 +356925.501}
SPL {X  -162.820, Y  +464.528, Z    +0.000, E1   +47.611, E3 +356941.715}
SPL {X  -162.820, Y  +458.830, Z    +0.000, E1   +46.994, E3 +356956.393}
SPL {X  -162.820, Y  +455.537, Z    +0.000, E1   +45.900, E3 +356969.212}
SPL {X  -162.820, Y  +452.032, Z    +0.000, E1   +45.224, E3 +356980.416}
SPL {X  -162.820, Y  +446.617, Z    +0.000, E1   +44.768, E3 +356994.503}
SPL {X  -162.820, Y  +440.464, Z    +0.000, E1   +44.845, E3 +357006.805}
SPL {X  -162.820, Y  +435.902, Z    +0.000, E1   +44.853, E3 +357016.328}
SPL {X  -162.820, Y  +429.336, Z    +0.000, E1   +44.917, E3 +357029.847}
SPL {X  -162.820, Y  +423.193, Z    +0.000, E1   +44.819, E3 +357043.106}
SPL {X  -162.820, Y  +416.810, Z    +0.000, E1   +44.932, E3 +357055.994}
SPL {X  -162.820, Y  +408.782, Z    +0.000, E1   +44.820, E3 +357073.424}
SPL {X  -162.820, Y  +401.619, Z    +0.000, E1   +44.978, E3 +357087.346}
SPL {X  -162.820, Y  +394.771, Z    +0.000, E1   +44.856, E3 +357102.585}
SPL {X  -162.820, Y  +387.883, Z    +0.000, E1   +44.837, E3 +357116.939}
SPL {X  -162.820, Y  +382.755, Z    +0.000, E1   +44.828, E3 +357127.732}
SPL {X  -162.796, Y  +377.700, Z    +0.000, E1   +44.829, E3 +357138.312}
SPL {X  -162.619, Y  +372.412, Z    +0.000, E1   +44.928, E3 +357148.772}
SPL {X  -162.311, Y  +367.633, Z    +0.000, E1   +44.798, E3 +357159.539}
SPL {X  -161.766, Y  +362.002, Z    +0.000, E1   +44.644, E3 +357172.297}
SPL {X  -161.043, Y  +356.508, Z    +0.000, E1   +44.528, E3 +357184.412}
SPL {X  -160.070, Y  +350.699, Z    +0.000, E1   +44.409, E3 +357197.364}
SPL {X  -158.853, Y  +344.776, Z    +0.000, E1   +44.148, E3 +357211.184}
SPL {X  -157.292, Y  +338.433, Z    +0.000, E1   +43.917, E3 +357225.863}
SPL {X  -155.654, Y  +332.729, Z    +0.000, E1   +43.534, E3 +357239.785}
SPL {X  -154.189, Y  +328.191, Z    +0.000, E1   +43.338, E3 +357250.281}
SPL {X  -149.333, Y  +315.614, Z    +0.000, E1   +46.650, E3 +357257.597}
SPL {X  -142.680, Y  +302.060, Z    +0.000, E1   +42.084, E3 +357323.941}
ENDSPLINE

SPLINE
SPL {X  -151.184, Y  +320.053, Z    +0.000, E1   +32.435, E3 +357391.184}
SPL {X  -158.917, Y  +345.064, Z    +0.000, E1   +21.858, E3 +357392.533}
SPL {X  -161.350, Y  +358.672, Z    +0.000, E1   +15.089, E3 +357395.235}
SPL {X  -162.491, Y  +370.147, Z    +0.000, E1    +8.815, E3 +357398.170}
SPL {X  -162.816, Y  +379.394, Z    +0.000, E1    +3.267, E3 +357397.998}
SPL {X  -162.820, Y  +384.427, Z    +0.000, E1    -0.390, E3 +357398.518}
SPL {X  -162.820, Y  +387.736, Z    +0.000, E1    -3.142, E3 +357397.798}
SPL {X  -162.820, Y  +391.456, Z    +0.000, E1    -6.603, E3 +357398.585}
SPL {X  -162.820, Y  +397.032, Z    +0.000, E1   -12.435, E3 +357398.032}
SPL {X  -162.820, Y  +406.111, Z    +0.000, E1   -22.010, E3 +357399.083}
SPL {X  -162.820, Y  +418.653, Z    +0.000, E1   -36.657, E3 +357393.436}
SPL {X  -162.820, Y  +440.590, Z    +0.000, E1   -50.152, E3 +357398.681}
SPL {X  -162.820, Y  +447.889, Z    +0.000, E1   -43.424, E3 +357429.827}
SPL {X  -162.820, Y  +478.087, Z    +0.000, E1   -45.903, E3 +357475.046}
ENDSPLINE

SPLINE
SPL {X  -162.820, Y  +474.900, Z    +0.000, E1   -42.394, E3 +357489.199}
ENDSPLINE

SPLINE
SPL {X  -162.820, Y  +480.895, Z    +0.000, E1   -42.223, E3 +357503.860}
SPL {X  -162.820, Y  +485.782, Z    +0.000, E1   -42.348, E3 +357514.206}
SPL {X  -162.820, Y  +489.480, Z    +0.000, E1   -42.230, E3 +357523.433}
SPL {X  -162.820, Y  +494.825, Z    +0.000, E1   -42.287, E3 +357535.380}
SPL {X  -162.820, Y  +501.023, Z    +0.000, E1   -42.347, E3 +357549.262}
SPL {X  -162.820, Y  +506.968, Z    +0.000, E1   -42.248, E3 +357563.453}
SPL {X  -162.820, Y  +513.215, Z    +0.000, E1   -42.304, E3 +357577.428}
SPL {X  -162.820, Y  +518.708, Z    +0.000, E1   -42.272, E3 +357590.149}
SPL {X  -162.820, Y  +525.147, Z    +0.000, E1   -42.298, E3 +357604.892}
SPL {X  -162.820, Y  +531.715, Z    +0.000, E1   -42.312, E3 +357619.717}
SPL {X  -162.820, Y  +537.459, Z    +0.000, E1   -42.308, E3 +357632.976}
SPL {X  -162.820, Y  +542.643, Z    +0.000, E1   -42.173, E3 +357645.569}
SPL {X  -162.820, Y  +549.160, Z    +0.000, E1   -42.387, E3 +357659.327}
SPL {X  -162.820, Y  +554.884, Z    +0.000, E1   -42.207, E3 +357673.413}
SPL {X  -162.820, Y  +561.114, Z    +0.000, E1   -42.336, E3 +357686.993}
SPL {X  -162.820, Y  +566.097, Z    +0.000, E1   -42.118, E3 +357699.603}
SPL {X  -162.820, Y  +571.654, Z    +0.000, E1   -42.313, E3 +357711.256}
SPL {X  -162.820, Y  +577.246, Z    +0.000, E1   -42.284, E3 +357724.222}
SPL {X  -162.820, Y  +582.233, Z    +0.000, E1   -42.188, E3 +357736.201}
SPL {X  -162.820, Y  +588.138, Z    +0.000, E1   -42.308, E3 +357749.100}
SPL {X  -162.820, Y  +593.999, Z    +0.000, E1   -42.301, E3 +357762.510}
SPL {X  -162.820, Y  +599.194, Z    +0.000, E1   -42.235, E3 +357774.814}
SPL {X  -162.820, Y  +604.595, Z    +0.000, E1   -42.290, E3 +357786.846}
SPL {X  -162.820, Y  +609.630, Z    +0.000, E1   -42.276, E3 +357798.472}
SPL {X  -162.820, Y  +614.392, Z    +0.000, E1   -42.242, E3 +357809.572}
SPL {X  -162.820, Y  +620.424, Z    +0.000, E1   -42.277, E3 +357823.319}
SPL {X  -162.820, Y  +626.430, Z    +0.000, E1   -42.291, E3 +357836.869}
SPL {X  -162.820, Y  +631.865, Z    +0.000, E1   -42.327, E3 +357849.163}
SPL {X  -162.820, Y  +637.189, Z    +0.000, E1   -42.236, E3 +357861.837}
SPL {X  -162.820, Y  +642.066, Z    +0.000, E1   -42.247, E3 +357872.959}
SPL {X  -162.820, Y  +646.907, Z    +0.000, E1   -42.249, E3 +357884.078}
SPL {X  -162.820, Y  +652.374, Z    +0.000, E1   -42.262, E3 +357896.516}
SPL {X  -162.820, Y  +657.439, Z    +0.000, E1   -42.251, E3 +357908.189}
SPL {X  -162.820, Y  +663.328, Z    +0.000, E1   -42.283, E3 +357921.591}
SPL {X  -162.820, Y  +669.078, Z    +0.000, E1   -42.263, E3 +357934.788}
SPL {X  -162.819, Y  +673.910, Z    +0.000, E1   -42.244, E3 +357945.982}
SPL {X  -162.729, Y  +678.944, Z    +0.000, E1   -42.273, E3 +357957.349}
SPL {X  -162.479, Y  +684.035, Z    +0.000, E1   -42.168, E3 +357969.687}
SPL {X  -162.026, Y  +689.560, Z    +0.000, E1   -42.192, E3 +357982.175}
SPL {X  -161.446, Y  +694.609, Z    +0.000, E1   -42.094, E3 +357994.307}
SPL {X  -160.889, Y  +698.503, Z    +0.000, E1   -41.849, E3 +358004.581}
SPL {X  -160.100, Y  +703.138, Z    +0.000, E1   -41.824, E3 +358015.440}
SPL {X  -158.994, Y  +708.588, Z    +0.000, E1   -41.616, E3 +358029.159}
SPL {X  -157.709, Y  +713.973, Z    +0.000, E1   -41.360, E3 +358042.941}
SPL {X  -156.530, Y  +718.319, Z    +0.000, E1   -41.164, E3 +358053.886}
SPL {X  -155.547, Y  +721.618, Z    +0.000, E1   -40.968, E3 +358062.510}
SPL {X  -151.388, Y  +733.433, Z    +0.000, E1   -44.269, E3 +358070.213}
SPL {X  -144.352, Y  +748.818, Z    +0.000, E1   -40.701, E3 +358139.247}
SPL {X  -143.859, Y  +749.757, Z    +0.000, E1   -39.148, E3 +358167.196}
ENDSPLINE

SPLINE
SPL {X  -159.245, Y  +707.432, Z    +0.000, E1   -21.244, E3 +358199.229}
SPL {X  -162.277, Y  +686.791, Z    +0.000, E1   -10.607, E3 +358200.639}
SPL {X  -162.766, Y  +677.687, Z    +0.000, E1    -5.239, E3 +358202.829}
SPL {X  -162.820, Y  +671.059, Z    +0.000, E1    -0.934, E3 +358203.185}
SPL {X  -162.820, Y  +665.599, Z    +0.000, E1    +3.424, E3 +358203.635}
SPL {X  -162.820, Y  +661.024, Z    +0.000, E1    +7.880, E3 +358203.103}
SPL {X  -162.820, Y  +654.280, Z    +0.000, E1   +14.617, E3 +358203.821}
SPL {X  -162.820, Y  +638.947, Z    +0.000, E1   +31.033, E3 +358201.874}
SPL {X  -162.820, Y  +608.150, Z    +0.000, E1   +43.921, E3 +358228.107}
SPL {X  -162.820, Y  +574.255, Z    +0.000, E1   +46.562, E3 +358277.901}
ENDSPLINE

SPLINE
SPL {X  -162.820, Y  +579.440, Z    +0.000, E1   +42.450, E3 +358291.088}
ENDSPLINE

SPLINE
SPL {X  -162.820, Y  +574.443, Z    +0.000, E1   +42.333, E3 +358303.183}
SPL {X  -162.820, Y  +568.554, Z    +0.000, E1   +42.362, E3 +358316.545}
SPL {X  -162.820, Y  +561.474, Z    +0.000, E1   +42.369, E3 +358332.731}
SPL {X  -162.820, Y  +555.861, Z    +0.000, E1   +42.349, E3 +358345.535}
SPL {X  -162.820, Y  +550.633, Z    +0.000, E1   +42.421, E3 +358357.065}
SPL {X  -162.820, Y  +546.534, Z    +0.000, E1   +42.268, E3 +358367.275}
SPL {X  -162.820, Y  +541.056, Z    +0.000, E1   +42.452, E3 +358378.790}
SPL {X  -162.820, Y  +535.223, Z    +0.000, E1   +42.386, E3 +358392.484}
SPL {X  -162.820, Y  +529.084, Z    +0.000, E1   +42.400, E3 +358406.406}
SPL {X  -162.820, Y  +522.568, Z    +0.000, E1   +42.385, E3 +358421.436}
SPL {X  -162.820, Y  +515.708, Z    +0.000, E1   +42.333, E3 +358437.404}
SPL {X  -162.820, Y  +510.265, Z    +0.000, E1   +42.390, E3 +358449.365}
SPL {X  -162.820, Y  +505.746, Z    +0.000, E1   +42.400, E3 +358459.678}
SPL {X  -162.820, Y  +500.461, Z    +0.000, E1   +42.387, E3 +358471.805}
SPL {X  -162.820, Y  +494.841, Z    +0.000, E1   +42.316, E3 +358485.131}
SPL {X  -162.820, Y  +487.903, Z    +0.000, E1   +42.488, E3 +358499.954}
SPL {X  -162.820, Y  +484.250, Z    +0.000, E1   +42.201, E3 +358509.815}
SPL {X  -162.820, Y  +464.528, Z    +0.000, E1   +47.611, E3 +358518.638}
SPL {X  -162.820, Y  +459.899, Z    +0.000, E1   +47.097, E3 +358530.480}
SPL {X  -162.820, Y  +455.990, Z    +0.000, E1   +46.212, E3 +358543.554}
SPL {X  -162.820, Y  +452.032, Z    +0.000, E1   +45.224, E3 +358557.340}
SPL {X  -162.820, Y  +446.617, Z    +0.000, E1   +44.768, E3 +358571.426}
SPL {X  -162.820, Y  +437.902, Z    +0.000, E1   +44.900, E3 +358589.003}
SPL {X  -162.820, Y  +430.894, Z    +0.000, E1   +44.976, E3 +358602.989}
SPL {X  -162.820, Y  +425.053, Z    +0.000, E1   +44.824, E3 +358616.250}
SPL {X  -162.820, Y  +418.403, Z    +0.000, E1   +44.941, E3 +358629.364}
SPL {X  -162.820, Y  +412.479, Z    +0.000, E1   +44.780, E3 +358642.794}
SPL {X  -162.820, Y  +406.707, Z    +0.000, E1   +44.849, E3 +358654.367}
SPL {X  -162.820, Y  +400.166, Z    +0.000, E1   +44.948, E3 +358667.651}
SPL {X  -162.820, Y  +393.279, Z    +0.000, E1   +44.825, E3 +358682.654}
SPL {X  -162.820, Y  +387.883, Z    +0.000, E1   +44.837, E3 +358693.862}
SPL {X  -162.820, Y  +382.755, Z    +0.000, E1   +44.828, E3 +358704.655}
SPL {X  -162.796, Y  +377.700, Z    +0.000, E1   +44.829, E3 +358715.235}
SPL {X  -162.619, Y  +372.412, Z    +0.000, E1   +44.928, E3 +358725.695}
SPL {X  -162.170, Y  +365.961, Z    +0.000, E1   +44.802, E3 +358740.124}
SPL {X  -161.259, Y  +358.011, Z    +0.000, E1   +44.581, E3 +358758.051}
SPL {X  -160.417, Y  +352.631, Z    +0.000, E1   +44.411, E3 +358770.066}
SPL {X  -159.784, Y  +349.204, Z    +0.000, E1   +44.340, E3 +358777.659}
SPL {X  -158.853, Y  +344.776, Z    +0.000, E1   +44.148, E3 +358788.107}
SPL {X  -157.292, Y  +338.433, Z    +0.000, E1   +43.917, E3 +358802.786}
SPL {X  -155.654, Y  +332.729, Z    +0.000, E1   +43.534, E3 +358816.708}
SPL {X  -154.189, Y  +328.191, Z    +0.000, E1   +43.338, E3 +358827.204}
SPL {X  -149.333, Y  +315.614, Z    +0.000, E1   +46.650, E3 +358834.520}
SPL {X  -142.680, Y  +302.060, Z    +0.000, E1   +42.084, E3 +358900.864}
ENDSPLINE

SPLINE
SPL {X  -151.184, Y  +320.053, Z    +0.000, E1   +32.435, E3 +358968.107}
SPL {X  -158.917, Y  +345.064, Z    +0.000, E1   +21.858, E3 +358969.456}
SPL {X  -161.350, Y  +358.672, Z    +0.000, E1   +15.089, E3 +358972.158}
SPL {X  -162.491, Y  +370.147, Z    +0.000, E1    +8.815, E3 +358975.093}
SPL {X  -162.771, Y  +376.522, Z    +0.000, E1    +5.005, E3 +358974.702}
SPL {X  -162.820, Y  +383.029, Z    +0.000, E1    +0.769, E3 +358975.270}
SPL {X  -162.820, Y  +387.736, Z    +0.000, E1    -3.142, E3 +358974.721}
SPL {X  -162.820, Y  +391.456, Z    +0.000, E1    -6.603, E3 +358975.508}
SPL {X  -162.820, Y  +397.032, Z    +0.000, E1   -12.435, E3 +358974.955}
SPL {X  -162.820, Y  +406.111, Z    +0.000, E1   -22.010, E3 +358976.006}
SPL {X  -162.820, Y  +418.653, Z    +0.000, E1   -36.657, E3 +358970.359}
SPL {X  -162.820, Y  +440.590, Z    +0.000, E1   -50.152, E3 +358975.604}
SPL {X  -162.820, Y  +447.889, Z    +0.000, E1   -43.424, E3 +359006.750}
SPL {X  -162.820, Y  +479.020, Z    +0.000, E1   -47.189, E3 +359046.327}
ENDSPLINE

SPLINE
SPL {X  -162.820, Y  +474.886, Z    +0.000, E1   -43.721, E3 +359058.211}
ENDSPLINE

SPLINE
SPL {X  -162.820, Y  +476.137, Z    +0.000, E1   -42.304, E3 +359069.324}
SPL {X  -162.820, Y  +480.895, Z    +0.000, E1   -42.223, E3 +359080.783}
SPL {X  -162.820, Y  +485.782, Z    +0.000, E1   -42.348, E3 +359091.129}
SPL {X  -162.820, Y  +489.480, Z    +0.000, E1   -42.230, E3 +359100.356}
SPL {X  -162.820, Y  +494.825, Z    +0.000, E1   -42.287, E3 +359112.303}
SPL {X  -162.820, Y  +501.909, Z    +0.000, E1   -42.324, E3 +359128.490}
SPL {X  -162.820, Y  +508.157, Z    +0.000, E1   -42.280, E3 +359142.820}
SPL {X  -162.820, Y  +513.215, Z    +0.000, E1   -42.304, E3 +359154.351}
SPL {X  -162.820, Y  +520.311, Z    +0.000, E1   -42.317, E3 +359170.649}
SPL {X  -162.820, Y  +526.529, Z    +0.000, E1   -42.247, E3 +359185.119}
SPL {X  -162.820, Y  +531.715, Z    +0.000, E1   -42.312, E3 +359196.641}
SPL {X  -162.820, Y  +537.459, Z    +0.000, E1   -42.308, E3 +359209.899}
SPL {X  -162.820, Y  +542.643, Z    +0.000, E1   -42.173, E3 +359222.492}
SPL {X  -162.820, Y  +549.160, Z    +0.000, E1   -42.387, E3 +359236.250}
SPL {X  -162.820, Y  +554.884, Z    +0.000, E1   -42.207, E3 +359250.336}
SPL {X  -162.820, Y  +561.114, Z    +0.000, E1   -42.336, E3 +359263.916}
SPL {X  -162.820, Y  +566.097, Z    +0.000, E1   -42.118, E3 +359276.526}
SPL {X  -162.820, Y  +571.654, Z    +0.000, E1   -42.313, E3 +359288.179}
SPL {X  -162.820, Y  +577.246, Z    +0.000, E1   -42.284, E3 +359301.145}
SPL {X  -162.820, Y  +582.233, Z    +0.000, E1   -42.188, E3 +359313.124}
SPL {X  -162.820, Y  +588.138, Z    +0.000, E1   -42.308, E3 +359326.023}
SPL {X  -162.820, Y  +593.999, Z    +0.000, E1   -42.301, E3 +359339.433}
SPL {X  -162.820, Y  +599.194, Z    +0.000, E1   -42.235, E3 +359351.737}
SPL {X  -162.820, Y  +604.595, Z    +0.000, E1   -42.290, E3 +359363.769}
SPL {X  -162.820, Y  +609.630, Z    +0.000, E1   -42.276, E3 +359375.395}
SPL {X  -162.820, Y  +614.392, Z    +0.000, E1   -42.242, E3 +359386.495}
SPL {X  -162.820, Y  +620.424, Z    +0.000, E1   -42.277, E3 +359400.243}
SPL {X  -162.820, Y  +626.430, Z    +0.000, E1   -42.291, E3 +359413.792}
SPL {X  -162.820, Y  +631.865, Z    +0.000, E1   -42.327, E3 +359426.086}
SPL {X  -162.820, Y  +637.189, Z    +0.000, E1   -42.236, E3 +359438.760}
SPL {X  -162.820, Y  +642.066, Z    +0.000, E1   -42.247, E3 +359449.882}
SPL {X  -162.820, Y  +646.907, Z    +0.000, E1   -42.249, E3 +359461.001}
SPL {X  -162.820, Y  +652.374, Z    +0.000, E1   -42.262, E3 +359473.439}
SPL {X  -162.820, Y  +657.439, Z    +0.000, E1   -42.251, E3 +359485.112}
SPL {X  -162.820, Y  +663.328, Z    +0.000, E1   -42.283, E3 +359498.514}
SPL {X  -162.820, Y  +669.078, Z    +0.000, E1   -42.263, E3 +359511.711}
SPL {X  -162.819, Y  +673.910, Z    +0.000, E1   -42.244, E3 +359522.905}
SPL {X  -162.729, Y  +678.944, Z    +0.000, E1   -42.273, E3 +359534.272}
SPL {X  -162.479, Y  +684.035, Z    +0.000, E1   -42.168, E3 +359546.610}
SPL {X  -162.026, Y  +689.560, Z    +0.000, E1   -42.192, E3 +359559.098}
SPL {X  -161.446, Y  +694.609, Z    +0.000, E1   -42.094, E3 +359571.230}
SPL {X  -160.681, Y  +699.806, Z    +0.000, E1   -41.866, E3 +359584.513}
SPL {X  -159.658, Y  +705.434, Z    +0.000, E1   -41.735, E3 +359598.143}
SPL {X  -158.502, Y  +710.748, Z    +0.000, E1   -41.532, E3 +359611.491}
SPL {X  -157.452, Y  +714.962, Z    +0.000, E1   -41.276, E3 +359622.486}
SPL {X  -156.530, Y  +718.319, Z    +0.000, E1   -41.164, E3 +359630.809}
SPL {X  -155.547, Y  +721.618, Z    +0.000, E1   -40.968, E3 +359639.433}
SPL {X  -151.388, Y  +733.433, Z    +0.000, E1   -44.269, E3 +359647.136}
SPL {X  -144.352, Y  +748.818, Z    +0.000, E1   -40.701, E3 +359716.171}
SPL {X  -143.859, Y  +749.757, Z    +0.000, E1   -39.148, E3 +359744.119}
ENDSPLINE

SPLINE
SPL {X  -159.245, Y  +707.432, Z    +0.000, E1   -21.244, E3 +359776.152}
SPL {X  -162.277, Y  +686.791, Z    +0.000, E1   -10.607, E3 +359777.562}
SPL {X  -162.766, Y  +677.687, Z    +0.000, E1    -5.239, E3 +359779.752}
SPL {X  -162.820, Y  +672.396, Z    +0.000, E1    -1.801, E3 +359780.541}
SPL {X  -162.820, Y  +667.851, Z    +0.000, E1    +1.551, E3 +359780.037}
SPL {X  -162.820, Y  +662.610, Z    +0.000, E1    +6.209, E3 +359780.411}
SPL {X  -162.820, Y  +654.280, Z    +0.000, E1   +14.617, E3 +359780.744}
SPL {X  -162.820, Y  +638.947, Z    +0.000, E1   +31.033, E3 +359778.797}
SPL {X  -162.820, Y  +608.150, Z    +0.000, E1   +43.921, E3 +359805.030}
SPL {X  -162.820, Y  +574.255, Z    +0.000, E1   +46.562, E3 +359854.824}
ENDSPLINE

SPLINE
SPL {X  -162.820, Y  +579.440, Z    +0.000, E1   +42.450, E3 +359868.012}
ENDSPLINE

SPLINE
SPL {X  -162.820, Y  +574.443, Z    +0.000, E1   +42.333, E3 +359880.106}
SPL {X  -162.820, Y  +568.554, Z    +0.000, E1   +42.362, E3 +359893.468}
SPL {X  -162.820, Y  +561.474, Z    +0.000, E1   +42.369, E3 +359909.654}
SPL {X  -162.820, Y  +555.861, Z    +0.000, E1   +42.349, E3 +359922.459}
SPL {X  -162.820, Y  +550.633, Z    +0.000, E1   +42.421, E3 +359933.989}
SPL {X  -162.820, Y  +546.534, Z    +0.000, E1   +42.268, E3 +359944.198}
SPL {X  -162.820, Y  +539.632, Z    +0.000, E1   +42.488, E3 +359958.919}
SPL {X  -162.820, Y  +533.959, Z    +0.000, E1   +42.310, E3 +359972.616}
SPL {X  -162.820, Y  +529.084, Z    +0.000, E1   +42.400, E3 +359983.330}
SPL {X  -162.820, Y  +524.911, Z    +0.000, E1   +42.325, E3 +359993.176}
SPL {X  -162.820, Y  +519.984, Z    +0.000, E1   +42.385, E3 +360004.246}
SPL {X  -162.820, Y  +512.536, Z    +0.000, E1   +42.385, E3 +360021.357}
SPL {X  -162.820, Y  +505.746, Z    +0.000, E1   +42.400, E3 +360036.601}
SPL {X  -162.820, Y  +500.461, Z    +0.000, E1   +42.387, E3 +360048.728}
SPL {X  -162.820, Y  +494.841, Z    +0.000, E1   +42.316, E3 +360062.055}
SPL {X  -162.820, Y  +489.758, Z    +0.000, E1   +42.464, E3 +360072.648}
SPL {X  -162.820, Y  +485.695, Z    +0.000, E1   +42.386, E3 +360082.484}
SPL {X  -162.820, Y  +464.528, Z    +0.000, E1   +47.611, E3 +360095.561}
SPL {X  -162.820, Y  +459.899, Z    +0.000, E1   +47.097, E3 +360107.403}
SPL {X  -162.820, Y  +455.990, Z    +0.000, E1   +46.212, E3 +360120.477}
SPL {X  -162.820, Y  +452.032, Z    +0.000, E1   +45.224, E3 +360134.263}
SPL {X  -162.820, Y  +446.617, Z    +0.000, E1   +44.768, E3 +360148.349}
SPL {X  -162.820, Y  +437.902, Z    +0.000, E1   +44.900, E3 +360165.926}
SPL {X  -162.820, Y  +429.336, Z    +0.000, E1   +44.917, E3 +360183.693}
SPL {X  -162.820, Y  +423.193, Z    +0.000, E1   +44.819, E3 +360196.952}
SPL {X  -162.820, Y  +418.403, Z    +0.000, E1   +44.941, E3 +360206.287}
SPL {X  -162.820, Y  +412.479, Z    +0.000, E1   +44.780, E3 +360219.717}
SPL {X  -162.820, Y  +406.707, Z    +0.000, E1   +44.849, E3 +360231.290}
SPL {X  -162.820, Y  +401.619, Z    +0.000, E1   +44.978, E3 +360241.192}
SPL {X  -162.820, Y  +394.771, Z    +0.000, E1   +44.856, E3 +360256.431}
SPL {X  -162.820, Y  +387.883, Z    +0.000, E1   +44.837, E3 +360270.785}
SPL {X  -162.820, Y  +382.755, Z    +0.000, E1   +44.828, E3 +360281.578}
SPL {X  -162.796, Y  +377.700, Z    +0.000, E1   +44.829, E3 +360292.158}
SPL {X  -162.619, Y  +372.412, Z    +0.000, E1   +44.928, E3 +360302.618}
SPL {X  -162.170, Y  +365.961, Z    +0.000, E1   +44.802, E3 +360317.047}
SPL {X  -161.259, Y  +358.011, Z    +0.000, E1   +44.581, E3 +360334.974}
SPL {X  -160.070, Y  +350.699, Z    +0.000, E1   +44.409, E3 +360351.210}
SPL {X  -158.853, Y  +344.776, Z    +0.000, E1   +44.148, E3 +360365.031}
SPL {X  -157.821, Y  +340.466, Z    +0.000, E1   +44.026, E3 +360374.623}
SPL {X  -156.950, Y  +337.174, Z    +0.000, E1   +43.768, E3 +360382.989}
SPL {X  -155.654, Y  +332.729, Z    +0.000, E1   +43.534, E3 +360393.631}
SPL {X  -154.189, Y  +328.191, Z    +0.000, E1   +43.338, E3 +360404.127}
SPL {X  -149.333, Y  +315.614, Z    +0.000, E1   +46.650, E3 +360411.443}
SPL {X  -142.680, Y  +302.060, Z    +0.000, E1   +42.084, E3 +360477.787}
ENDSPLINE

SPLINE
SPL {X  -151.184, Y  +320.053, Z    +0.000, E1   +32.435, E3 +360545.030}
SPL {X  -158.917, Y  +345.064, Z    +0.000, E1   +21.858, E3 +360546.379}
SPL {X  -161.350, Y  +358.672, Z    +0.000, E1   +15.089, E3 +360549.082}
SPL {X  -162.491, Y  +370.147, Z    +0.000, E1    +8.815, E3 +360552.016}
SPL {X  -162.816, Y  +379.394, Z    +0.000, E1    +3.267, E3 +360551.844}
SPL {X  -162.820, Y  +384.427, Z    +0.000, E1    -0.390, E3 +360552.364}
SPL {X  -162.820, Y  +387.736, Z    +0.000, E1    -3.142, E3 +360551.644}
SPL {X  -162.820, Y  +391.456, Z    +0.000, E1    -6.603, E3 +360552.431}
SPL {X  -162.820, Y  +397.032, Z    +0.000, E1   -12.435, E3 +360551.878}
SPL {X  -162.820, Y  +406.111, Z    +0.000, E1   -22.010, E3 +360552.929}
SPL {X  -162.820, Y  +418.653, Z    +0.000, E1   -36.657, E3 +360547.282}
SPL {X  -162.820, Y  +440.590, Z    +0.000, E1   -50.152, E3 +360552.528}
SPL {X  -162.820, Y  +447.889, Z    +0.000, E1   -43.424, E3 +360583.673}
SPL {X  -162.820, Y  +478.087, Z    +0.000, E1   -45.903, E3 +360628.892}
ENDSPLINE

SPLINE
SPL {X  -162.820, Y  +472.818, Z    +0.000, E1   -42.437, E3 +360637.833}
ENDSPLINE

SPLINE
SPL {X  -162.820, Y  +477.319, Z    +0.000, E1   -42.306, E3 +360649.060}
SPL {X  -162.820, Y  +483.923, Z    +0.000, E1   -42.291, E3 +360664.267}
SPL {X  -162.820, Y  +489.480, Z    +0.000, E1   -42.230, E3 +360677.279}
SPL {X  -162.820, Y  +494.825, Z    +0.000, E1   -42.287, E3 +360689.226}
SPL {X  -162.820, Y  +501.023, Z    +0.000, E1   -42.347, E3 +360703.109}
SPL {X  -162.820, Y  +506.968, Z    +0.000, E1   -42.248, E3 +360717.300}
SPL {X  -162.820, Y  +513.215, Z    +0.000, E1   -42.304, E3 +360731.274}
SPL {X  -162.820, Y  +518.708, Z    +0.000, E1   -42.272, E3 +360743.995}
SPL {X  -162.820, Y  +525.147, Z    +0.000, E1   -42.298, E3 +360758.738}
SPL {X  -162.820, Y  +531.715, Z    +0.000, E1   -42.312, E3 +360773.564}
SPL {X  -162.820, Y  +537.459, Z    +0.000, E1   -42.308, E3 +360786.823}
SPL {X  -162.820, Y  +542.643, Z    +0.000, E1   -42.173, E3 +360799.415}
SPL {X  -162.820, Y  +549.160, Z    +0.000, E1   -42.387, E3 +360813.173}
SPL {X  -162.820, Y  +554.884, Z    +0.000, E1   -42.207, E3 +360827.259}
SPL {X  -162.820, Y  +561.114, Z    +0.000, E1   -42.336, E3 +360840.839}
SPL {X  -162.820, Y  +566.097, Z    +0.000, E1   -42.118, E3 +360853.449}
SPL {X  -162.820, Y  +571.654, Z    +0.000, E1   -42.313, E3 +360865.103}
SPL {X  -162.820, Y  +577.246, Z    +0.000, E1   -42.284, E3 +360878.068}
SPL {X  -162.820, Y  +583.926, Z    +0.000, E1   -42.266, E3 +360893.628}
SPL {X  -162.820, Y  +589.581, Z    +0.000, E1   -42.277, E3 +360906.305}
SPL {X  -162.820, Y  +593.999, Z    +0.000, E1   -42.301, E3 +360916.356}
SPL {X  -162.820, Y  +599.194, Z    +0.000, E1   -42.235, E3 +360928.660}
SPL {X  -162.820, Y  +604.595, Z    +0.000, E1   -42.290, E3 +360940.692}
SPL {X  -162.820, Y  +609.630, Z    +0.000, E1   -42.276, E3 +360952.318}
SPL {X  -162.820, Y  +614.392, Z    +0.000, E1   -42.242, E3 +360963.418}
SPL {X  -162.820, Y  +620.424, Z    +0.000, E1   -42.277, E3 +360977.166}
SPL {X  -162.820, Y  +626.430, Z    +0.000, E1   -42.291, E3 +360990.715}
SPL {X  -162.820, Y  +631.865, Z    +0.000, E1   -42.327, E3 +361003.009}
SPL {X  -162.820, Y  +637.189, Z    +0.000, E1   -42.236, E3 +361015.683}
SPL {X  -162.820, Y  +642.066, Z    +0.000, E1   -42.247, E3 +361026.805}
SPL {X  -162.820, Y  +646.907, Z    +0.000, E1   -42.249, E3 +361037.924}
SPL {X  -162.820, Y  +652.374, Z    +0.000, E1   -42.262, E3 +361050.362}
SPL {X  -162.820, Y  +657.439, Z    +0.000, E1   -42.251, E3 +361062.035}
SPL {X  -162.820, Y  +663.328, Z    +0.000, E1   -42.283, E3 +361075.437}
SPL {X  -162.820, Y  +669.078, Z    +0.000, E1   -42.263, E3 +361088.634}
SPL {X  -162.819, Y  +673.910, Z    +0.000, E1   -42.244, E3 +361099.828}
SPL {X  -162.729, Y  +678.944, Z    +0.000, E1   -42.273, E3 +361111.195}
SPL {X  -162.479, Y  +684.035, Z    +0.000, E1   -42.168, E3 +361123.533}
SPL {X  -162.026, Y  +689.560, Z    +0.000, E1   -42.192, E3 +361136.021}
SPL {X  -161.446, Y  +694.609, Z    +0.000, E1   -42.094, E3 +361148.153}
SPL {X  -160.889, Y  +698.503, Z    +0.000, E1   -41.849, E3 +361158.427}
SPL {X  -159.869, Y  +704.360, Z    +0.000, E1   -41.806, E3 +361172.369}
SPL {X  -158.502, Y  +710.748, Z    +0.000, E1   -41.532, E3 +361188.414}
SPL {X  -156.963, Y  +716.777, Z    +0.000, E1   -41.265, E3 +361203.836}
SPL {X  -155.547, Y  +721.618, Z    +0.000, E1   -40.968, E3 +361216.356}
SPL {X  -151.388, Y  +733.433, Z    +0.000, E1   -44.269, E3 +361224.059}
SPL {X  -144.352, Y  +748.818, Z    +0.000, E1   -40.701, E3 +361293.094}
SPL {X  -143.859, Y  +749.757, Z    +0.000, E1   -39.148, E3 +361321.042}
ENDSPLINE

SPLINE
SPL {X  -159.245, Y  +707.432, Z    +0.000, E1   -21.244, E3 +361353.075}
SPL {X  -162.277, Y  +686.791, Z    +0.000, E1   -10.607, E3 +361354.485}
SPL {X  -162.766, Y  +677.687, Z    +0.000, E1    -5.239, E3 +361356.675}
SPL {X  -162.820, Y  +672.396, Z    +0.000, E1    -1.801, E3 +361357.464}
SPL {X  -162.820, Y  +667.851, Z    +0.000, E1    +1.551, E3 +361356.960}
SPL {X  -162.820, Y  +662.610, Z    +0.000, E1    +6.209, E3 +361357.334}
SPL {X  -162.820, Y  +654.280, Z    +0.000, E1   +14.617, E3 +361357.667}
SPL {X  -162.820, Y  +638.947, Z    +0.000, E1   +31.033, E3 +361355.720}
SPL {X  -162.820, Y  +608.150, Z    +0.000, E1   +43.921, E3 +361381.953}
SPL {X  -162.820, Y  +574.255, Z    +0.000, E1   +46.562, E3 +361431.747}
ENDSPLINE

SPLINE
SPL {X  -162.820, Y  +579.440, Z    +0.000, E1   +42.450, E3 +361444.935}
ENDSPLINE

SPLINE
SPL {X  -162.820, Y  +573.350, Z    +0.000, E1   +42.340, E3 +361459.612}
SPL {X  -162.820, Y  +565.899, Z    +0.000, E1   +42.413, E3 +361476.196}
SPL {X  -162.820, Y  +560.278, Z    +0.000, E1   +42.308, E3 +361489.533}
SPL {X  -162.820, Y  +555.861, Z    +0.000, E1   +42.349, E3 +361499.382}
SPL {X  -162.820, Y  +550.633, Z    +0.000, E1   +42.421, E3 +361510.912}
SPL {X  -162.820, Y  +546.534, Z    +0.000, E1   +42.268, E3 +361521.121}
SPL {X  -162.820, Y  +539.632, Z    +0.000, E1   +42.488, E3 +361535.842}
SPL {X  -162.820, Y  +533.959, Z    +0.000, E1   +42.310, E3 +361549.539}
SPL {X  -162.820, Y  +527.661, Z    +0.000, E1   +42.425, E3 +361563.535}
SPL {X  -162.820, Y  +521.246, Z    +0.000, E1   +42.365, E3 +361578.287}
SPL {X  -162.820, Y  +515.708, Z    +0.000, E1   +42.333, E3 +361591.250}
SPL {X  -162.820, Y  +510.265, Z    +0.000, E1   +42.390, E3 +361603.212}
SPL {X  -162.820, Y  +505.746, Z    +0.000, E1   +42.400, E3 +361613.524}
SPL {X  -162.820, Y  +500.461, Z    +0.000, E1   +42.387, E3 +361625.651}
SPL {X  -162.820, Y  +494.841, Z    +0.000, E1   +42.316, E3 +361638.978}
SPL {X  -162.820, Y  +486.958, Z    +0.000, E1   +42.460, E3 +361656.271}
SPL {X  -162.820, Y  +464.528, Z    +0.000, E1   +47.611, E3 +361672.484}
SPL {X  -162.820, Y  +458.830, Z    +0.000, E1   +46.994, E3 +361687.162}
SPL {X  -162.820, Y  +455.537, Z    +0.000, E1   +45.900, E3 +361699.981}
SPL {X  -162.820, Y  +452.032, Z    +0.000, E1   +45.224, E3 +361711.186}
SPL {X  -162.820, Y  +446.617, Z    +0.000, E1   +44.768, E3 +361725.272}
SPL {X  -162.820, Y  +440.464, Z    +0.000, E1   +44.845, E3 +361737.574}
SPL {X  -162.820, Y  +435.902, Z    +0.000, E1   +44.853, E3 +361747.098}
SPL {X  -162.820, Y  +429.336, Z    +0.000, E1   +44.917, E3 +361760.616}
SPL {X  -162.820, Y  +423.193, Z    +0.000, E1   +44.819, E3 +361773.875}
SPL {X  -162.820, Y  +418.403, Z    +0.000, E1   +44.941, E3 +361783.210}
SPL {X  -162.820, Y  +412.479, Z    +0.000, E1   +44.780, E3 +361796.640}
SPL {X  -162.820, Y  +406.707, Z    +0.000, E1   +44.849, E3 +361808.213}
SPL {X  -162.820, Y  +400.166, Z    +0.000, E1   +44.948, E3 +361821.497}
SPL {X  -162.820, Y  +393.279, Z    +0.000, E1   +44.825, E3 +361836.500}
SPL {X  -162.820, Y  +387.883, Z    +0.000, E1   +44.837, E3 +361847.708}
SPL {X  -162.820, Y  +382.755, Z    +0.000, E1   +44.828, E3 +361858.501}
SPL {X  -162.796, Y  +377.700, Z    +0.000, E1   +44.829, E3 +361869.081}
SPL {X  -162.619, Y  +372.412, Z    +0.000, E1   +44.928, E3 +361879.541}
SPL {X  -162.311, Y  +367.633, Z    +0.000, E1   +44.798, E3 +361890.308}
SPL {X  -161.766, Y  +362.002, Z    +0.000, E1   +44.644, E3 +361903.067}
SPL {X  -161.043, Y  +356.508, Z    +0.000, E1   +44.528, E3 +361915.181}
SPL {X  -160.417, Y  +352.631, Z    +0.000, E1   +44.411, E3 +361923.912}
SPL {X  -159.536, Y  +347.962, Z    +0.000, E1   +44.302, E3 +361934.439}
SPL {X  -158.195, Y  +341.969, Z    +0.000, E1   +44.082, E3 +361948.221}
SPL {X  -156.950, Y  +337.174, Z    +0.000, E1   +43.768, E3 +361959.912}
SPL {X  -155.654, Y  +332.729, Z    +0.000, E1   +43.534, E3 +361970.554}
SPL {X  -153.067, Y  +324.996, Z    +0.000, E1   +44.257, E3 +361982.608}
SPL {X  -147.786, Y  +312.164, Z    +0.000, E1   +47.292, E3 +361991.338}
SPL {X  -142.680, Y  +302.060, Z    +0.000, E1   +42.084, E3 +362054.710}
ENDSPLINE

SPLINE
SPL {X  -151.184, Y  +320.053, Z    +0.000, E1   +32.435, E3 +362121.954}
SPL {X  -158.917, Y  +345.064, Z    +0.000, E1   +21.858, E3 +362123.302}
SPL {X  -161.350, Y  +358.672, Z    +0.000, E1   +15.089, E3 +362126.005}
SPL {X  -162.491, Y  +370.147, Z    +0.000, E1    +8.815, E3 +362128.939}
SPL {X  -162.816, Y  +379.394, Z    +0.000, E1    +3.267, E3 +362128.767}
SPL {X  -162.820, Y  +384.427, Z    +0.000, E1    -0.390, E3 +362129.287}
SPL {X  -162.820, Y  +387.736, Z    +0.000, E1    -3.142, E3 +362128.567}
SPL {X  -162.820, Y  +392.770, Z    +0.000, E1    -7.830, E3 +362129.219}
SPL {X  -162.820, Y  +398.469, Z    +0.000, E1   -14.078, E3 +362128.672}
SPL {X  -162.820, Y  +406.111, Z    +0.000, E1   -22.010, E3 +362129.852}
SPL {X  -162.820, Y  +418.653, Z    +0.000, E1   -36.657, E3 +362124.205}
SPL {X  -162.820, Y  +440.590, Z    +0.000, E1   -50.152, E3 +362129.451}
SPL {X  -162.820, Y  +447.889, Z    +0.000, E1   -43.424, E3 +362160.596}
SPL {X  -162.820, Y  +479.020, Z    +0.000, E1   -47.189, E3 +362200.173}
ENDSPLINE

SPLINE
SPL {X  -162.820, Y  +474.886, Z    +0.000, E1   -43.721, E3 +362212.057}
ENDSPLINE

SPLINE
SPL {X  -162.820, Y  +477.319, Z    +0.000, E1   -42.306, E3 +362225.983}
SPL {X  -162.820, Y  +483.923, Z    +0.000, E1   -42.291, E3 +362241.190}
SPL {X  -162.820, Y  +489.480, Z    +0.000, E1   -42.230, E3 +362254.202}
SPL {X  -162.820, Y  +494.825, Z    +0.000, E1   -42.287, E3 +362266.150}
SPL {X  -162.820, Y  +501.023, Z    +0.000, E1   -42.347, E3 +362280.032}
SPL {X  -162.820, Y  +506.968, Z    +0.000, E1   -42.248, E3 +362294.223}
SPL {X  -162.820, Y  +513.215, Z    +0.000, E1   -42.304, E3 +362308.197}
SPL {X  -162.820, Y  +518.708, Z    +0.000, E1   -42.272, E3 +362320.919}
SPL {X  -162.820, Y  +525.147, Z    +0.000, E1   -42.298, E3 +362335.661}
SPL {X  -162.820, Y  +531.715, Z    +0.000, E1   -42.312, E3 +362350.487}
SPL {X  -162.820, Y  +537.459, Z    +0.000, E1   -42.308, E3 +362363.746}
SPL {X  -162.820, Y  +542.643, Z    +0.000, E1   -42.173, E3 +362376.338}
SPL {X  -162.820, Y  +549.160, Z    +0.000, E1   -42.387, E3 +362390.096}
SPL {X  -162.820, Y  +554.884, Z    +0.000, E1   -42.207, E3 +362404.182}
SPL {X  -162.820, Y  +561.114, Z    +0.000, E1   -42.336, E3 +362417.762}
SPL {X  -162.820, Y  +566.097, Z    +0.000, E1   -42.118, E3 +362430.372}
SPL {X  -162.820, Y  +571.654, Z    +0.000, E1   -42.313, E3 +362442.026}
SPL {X  -162.820, Y  +577.246, Z    +0.000, E1   -42.284, E3 +362454.991}
SPL {X  -162.820, Y  +582.233, Z    +0.000, E1   -42.188, E3 +362466.970}
SPL {X  -162.820, Y  +588.138, Z    +0.000, E1   -42.308, E3 +362479.869}
SPL {X  -162.820, Y  +593.999, Z    +0.000, E1   -42.301, E3 +362493.279}
SPL {X  -162.820, Y  +599.194, Z    +0.000, E1   -42.235, E3 +362505.584}
SPL {X  -162.820, Y  +604.595, Z    +0.000, E1   -42.290, E3 +362517.615}
SPL {X  -162.820, Y  +609.630, Z    +0.000, E1   -42.276, E3 +362529.241}
SPL {X  -162.820, Y  +614.392, Z    +0.000, E1   -42.242, E3 +362540.341}
SPL {X  -162.820, Y  +620.424, Z    +0.000, E1   -42.277, E3 +362554.089}
SPL {X  -162.820, Y  +626.430, Z    +0.000, E1   -42.291, E3 +362567.638}
SPL {X  -162.820, Y  +631.865, Z    +0.000, E1   -42.327, E3 +362579.932}
SPL {X  -162.820, Y  +637.189, Z    +0.000, E1   -42.236, E3 +362592.606}
SPL {X  -162.820, Y  +642.066, Z    +0.000, E1   -42.247, E3 +362603.728}
SPL {X  -162.820, Y  +646.907, Z    +0.000, E1   -42.249, E3 +362614.847}
SPL {X  -162.820, Y  +652.374, Z    +0.000, E1   -42.262, E3 +362627.286}
SPL {X  -162.820, Y  +658.634, Z    +0.000, E1   -42.281, E3 +362641.643}
SPL {X  -162.820, Y  +664.480, Z    +0.000, E1   -42.257, E3 +362655.037}
SPL {X  -162.820, Y  +669.078, Z    +0.000, E1   -42.263, E3 +362665.557}
SPL {X  -162.819, Y  +673.910, Z    +0.000, E1   -42.244, E3 +362676.751}
SPL {X  -162.729, Y  +678.944, Z    +0.000, E1   -42.273, E3 +362688.119}
SPL {X  -162.479, Y  +684.035, Z    +0.000, E1   -42.168, E3 +362700.456}
SPL {X  -162.026, Y  +689.560, Z    +0.000, E1   -42.192, E3 +362712.945}
SPL {X  -161.446, Y  +694.609, Z    +0.000, E1   -42.094, E3 +362725.077}
SPL {X  -160.681, Y  +699.806, Z    +0.000, E1   -41.866, E3 +362738.360}
SPL {X  -159.658, Y  +705.434, Z    +0.000, E1   -41.735, E3 +362751.990}
SPL {X  -158.502, Y  +710.748, Z    +0.000, E1   -41.532, E3 +362765.337}
SPL {X  -157.452, Y  +714.962, Z    +0.000, E1   -41.276, E3 +362776.332}
SPL {X  -156.530, Y  +718.319, Z    +0.000, E1   -41.164, E3 +362784.655}
SPL {X  -155.547, Y  +721.618, Z    +0.000, E1   -40.968, E3 +362793.279}
SPL {X  -151.388, Y  +733.433, Z    +0.000, E1   -44.269, E3 +362800.982}
SPL {X  -144.352, Y  +748.818, Z    +0.000, E1   -40.701, E3 +362870.017}
SPL {X  -143.859, Y  +749.757, Z    +0.000, E1   -39.148, E3 +362897.965}
ENDSPLINE

SPLINE
SPL {X  -159.245, Y  +707.432, Z    +0.000, E1   -21.244, E3 +362929.998}
SPL {X  -162.277, Y  +686.791, Z    +0.000, E1   -10.607, E3 +362931.408}
SPL {X  -162.766, Y  +677.687, Z    +0.000, E1    -5.239, E3 +362933.598}
SPL {X  -162.820, Y  +671.059, Z    +0.000, E1    -0.934, E3 +362933.954}
SPL {X  -162.820, Y  +666.960, Z    +0.000, E1    +2.343, E3 +362934.231}
SPL {X  -162.820, Y  +662.610, Z    +0.000, E1    +6.209, E3 +362934.257}
SPL {X  -162.820, Y  +654.280, Z    +0.000, E1   +14.617, E3 +362934.590}
SPL {X  -162.820, Y  +638.947, Z    +0.000, E1   +31.033, E3 +362932.643}
SPL {X  -162.820, Y  +608.150, Z    +0.000, E1   +43.921, E3 +362958.876}
SPL {X  -162.820, Y  +574.255, Z    +0.000, E1   +46.562, E3 +363008.670}
ENDSPLINE

SPLINE
SPL {X  -162.820, Y  +579.440, Z    +0.000, E1   +42.450, E3 +363021.858}
ENDSPLINE

SPLINE
SPL {X  -162.820, Y  +574.443, Z    +0.000, E1   +42.333, E3 +363033.952}
SPL {X  -162.820, Y  +568.554, Z    +0.000, E1   +42.362, E3 +363047.315}
SPL {X  -162.820, Y  +561.474, Z    +0.000, E1   +42.369, E3 +363063.500}
SPL {X  -162.820, Y  +554.421, Z    +0.000, E1   +42.414, E3 +363079.324}
SPL {X  -162.820, Y  +547.774, Z    +0.000, E1   +42.344, E3 +363094.898}
SPL {X  -162.820, Y  +541.056, Z    +0.000, E1   +42.452, E3 +363109.559}
SPL {X  -162.820, Y  +535.223, Z    +0.000, E1   +42.386, E3 +363123.253}
SPL {X  -162.820, Y  +529.084, Z    +0.000, E1   +42.400, E3 +363137.176}
SPL {X  -162.820, Y  +522.568, Z    +0.000, E1   +42.385, E3 +363152.205}
SPL {X  -162.820, Y  +515.708, Z    +0.000, E1   +42.333, E3 +363168.173}
SPL {X  -162.820, Y  +508.859, Z    +0.000, E1   +42.416, E3 +363183.315}
SPL {X  -162.820, Y  +501.651, Z    +0.000, E1   +42.423, E3 +363199.791}
SPL {X  -162.820, Y  +494.841, Z    +0.000, E1   +42.316, E3 +363215.901}
SPL {X  -162.820, Y  +486.958, Z    +0.000, E1   +42.460, E3 +363233.194}
SPL {X  -162.820, Y  +466.305, Z    +0.000, E1   +47.564, E3 +363246.201}
SPL {X  -162.820, Y  +460.790, Z    +0.000, E1   +47.323, E3 +363258.376}
SPL {X  -162.820, Y  +455.990, Z    +0.000, E1   +46.212, E3 +363274.324}
SPL {X  -162.820, Y  +452.032, Z    +0.000, E1   +45.224, E3 +363288.109}
SPL {X  -162.820, Y  +446.617, Z    +0.000, E1   +44.768, E3 +363302.195}
SPL {X  -162.820, Y  +437.902, Z    +0.000, E1   +44.900, E3 +363319.772}
SPL {X  -162.820, Y  +430.894, Z    +0.000, E1   +44.976, E3 +363333.758}
SPL {X  -162.820, Y  +425.053, Z    +0.000, E1   +44.824, E3 +363347.020}
SPL {X  -162.820, Y  +416.810, Z    +0.000, E1   +44.932, E3 +363363.686}
SPL {X  -162.820, Y  +408.782, Z    +0.000, E1   +44.820, E3 +363381.117}
SPL {X  -162.820, Y  +401.619, Z    +0.000, E1   +44.978, E3 +363395.038}
SPL {X  -162.820, Y  +394.771, Z    +0.000, E1   +44.856, E3 +363410.277}
SPL {X  -162.820, Y  +387.883, Z    +0.000, E1   +44.837, E3 +363424.631}
SPL {X  -162.820, Y  +382.755, Z    +0.000, E1   +44.828, E3 +363435.424}
SPL {X  -162.796, Y  +377.700, Z    +0.000, E1   +44.829, E3 +363446.004}
SPL {X  -162.619, Y  +372.412, Z    +0.000, E1   +44.928, E3 +363456.464}
SPL {X  -162.311, Y  +367.633, Z    +0.000, E1   +44.798, E3 +363467.231}
SPL {X  -161.766, Y  +362.002, Z    +0.000, E1   +44.644, E3 +363479.990}
SPL {X  -161.043, Y  +356.508, Z    +0.000, E1   +44.528, E3 +363492.104}
SPL {X  -160.070, Y  +350.699, Z    +0.000, E1   +44.409, E3 +363505.056}
SPL {X  -158.853, Y  +344.776, Z    +0.000, E1   +44.148, E3 +363518.877}
SPL {X  -157.292, Y  +338.433, Z    +0.000, E1   +43.917, E3 +363533.555}
SPL {X  -155.654, Y  +332.729, Z    +0.000, E1   +43.534, E3 +363547.477}
SPL {X  -154.189, Y  +328.191, Z    +0.000, E1   +43.338, E3 +363557.973}
SPL {X  -149.333, Y  +315.614, Z    +0.000, E1   +46.650, E3 +363565.289}
SPL {X  -142.680, Y  +302.060, Z    +0.000, E1   +42.084, E3 +363631.634}
ENDSPLINE

SPLINE
SPL {X  -151.184, Y  +320.053, Z    +0.000, E1   +32.435, E3 +363698.877}
SPL {X  -158.917, Y  +345.064, Z    +0.000, E1   +21.858, E3 +363700.225}
SPL {X  -161.350, Y  +358.672, Z    +0.000, E1   +15.089, E3 +363702.928}
SPL {X  -162.491, Y  +370.147, Z    +0.000, E1    +8.815, E3 +363705.862}
SPL {X  -162.771, Y  +376.522, Z    +0.000, E1    +5.005, E3 +363705.472}
SPL {X  -162.820, Y  +383.029, Z    +0.000, E1    +0.769, E3 +363706.039}
SPL {X  -162.820, Y  +387.736, Z    +0.000, E1    -3.142, E3 +363705.490}
SPL {X  -162.820, Y  +392.770, Z    +0.000, E1    -7.830, E3 +363706.142}
SPL {X  -162.820, Y  +398.469, Z    +0.000, E1   -14.078, E3 +363705.595}
SPL {X  -162.820, Y  +406.111, Z    +0.000, E1   -22.010, E3 +363706.775}
SPL {X  -162.820, Y  +418.653, Z    +0.000, E1   -36.657, E3 +363701.128}
SPL {X  -162.820, Y  +440.590, Z    +0.000, E1   -50.152, E3 +363706.374}
SPL {X  -162.820, Y  +447.889, Z    +0.000, E1   -43.424, E3 +363737.520}
SPL {X  -162.820, Y  +478.087, Z    +0.000, E1   -45.903, E3 +363782.739}
ENDSPLINE

SPLINE
SPL {X  -162.820, Y  +474.900, Z    +0.000, E1   -42.394, E3 +363796.891}
ENDSPLINE

SPLINE
SPL {X  -162.820, Y  +480.895, Z    +0.000, E1   -42.223, E3 +363811.553}
SPL {X  -162.820, Y  +485.782, Z    +0.000, E1   -42.348, E3 +363821.898}
SPL {X  -162.820, Y  +489.480, Z    +0.000, E1   -42.230, E3 +363831.125}
SPL {X  -162.820, Y  +494.825, Z    +0.000, E1   -42.287, E3 +363843.073}
SPL {X  -162.820, Y  +501.023, Z    +0.000, E1   -42.347, E3 +363856.955}
SPL {X  -162.820, Y  +506.968, Z    +0.000, E1   -42.248, E3 +363871.146}
SPL {X  -162.820, Y  +513.215, Z    +0.000, E1   -42.304, E3 +363885.120}
SPL {X  -162.820, Y  +518.708, Z    +0.000, E1   -42.272, E3 +363897.842}
SPL {X  -162.820, Y  +525.147, Z    +0.000, E1   -42.298, E3 +363912.584}
SPL {X  -162.820, Y  +531.715, Z    +0.000, E1   -42.312, E3 +363927.410}
SPL {X  -162.820, Y  +537.459, Z    +0.000, E1   -42.308, E3 +363940.669}
SPL {X  -162.820, Y  +542.643, Z    +0.000, E1   -42.173, E3 +363953.261}
SPL {X  -162.820, Y  +549.160, Z    +0.000, E1   -42.387, E3 +363967.019}
SPL {X  -162.820, Y  +554.884, Z    +0.000, E1   -42.207, E3 +363981.105}
SPL {X  -162.820, Y  +561.114, Z    +0.000, E1   -42.336, E3 +363994.685}
SPL {X  -162.820, Y  +566.097, Z    +0.000, E1   -42.118, E3 +364007.296}
SPL {X  -162.820, Y  +571.654, Z    +0.000, E1   -42.313, E3 +364018.949}
SPL {X  -162.820, Y  +577.246, Z    +0.000, E1   -42.284, E3 +364031.914}
SPL {X  -162.820, Y  +582.233, Z    +0.000, E1   -42.188, E3 +364043.893}
SPL {X  -162.820, Y  +588.138, Z    +0.000, E1   -42.308, E3 +364056.792}
SPL {X  -162.820, Y  +593.999, Z    +0.000, E1   -42.301, E3 +364070.202}
SPL {X  -162.820, Y  +599.194, Z    +0.000, E1   -42.235, E3 +364082.507}
SPL {X  -162.820, Y  +604.595, Z    +0.000, E1   -42.290, E3 +364094.538}
SPL {X  -162.820, Y  +609.630, Z    +0.000, E1   -42.276, E3 +364106.164}
SPL {X  -162.820, Y  +614.392, Z    +0.000, E1   -42.242, E3 +364117.264}
SPL {X  -162.820, Y  +620.424, Z    +0.000, E1   -42.277, E3 +364131.012}
SPL {X  -162.820, Y  +626.430, Z    +0.000, E1   -42.291, E3 +364144.561}
SPL {X  -162.820, Y  +631.865, Z    +0.000, E1   -42.327, E3 +364156.855}
SPL {X  -162.820, Y  +637.189, Z    +0.000, E1   -42.236, E3 +364169.529}
SPL {X  -162.820, Y  +642.066, Z    +0.000, E1   -42.247, E3 +364180.651}
SPL {X  -162.820, Y  +646.907, Z    +0.000, E1   -42.249, E3 +364191.770}
SPL {X  -162.820, Y  +652.374, Z    +0.000, E1   -42.262, E3 +364204.209}
SPL {X  -162.820, Y  +657.439, Z    +0.000, E1   -42.251, E3 +364215.882}
SPL {X  -162.820, Y  +663.328, Z    +0.000, E1   -42.283, E3 +364229.284}
SPL {X  -162.820, Y  +669.078, Z    +0.000, E1   -42.263, E3 +364242.480}
SPL {X  -162.819, Y  +673.910, Z    +0.000, E1   -42.244, E3 +364253.674}
SPL {X  -162.729, Y  +678.944, Z    +0.000, E1   -42.273, E3 +364265.042}
SPL {X  -162.479, Y  +684.035, Z    +0.000, E1   -42.168, E3 +364277.379}
SPL {X  -162.026, Y  +689.560, Z    +0.000, E1   -42.192, E3 +364289.868}
SPL {X  -161.446, Y  +694.609, Z    +0.000, E1   -42.094, E3 +364302.000}
SPL {X  -160.889, Y  +698.503, Z    +0.000, E1   -41.849, E3 +364312.274}
SPL {X  -160.100, Y  +703.138, Z    +0.000, E1   -41.824, E3 +364323.132}
SPL {X  -158.994, Y  +708.588, Z    +0.000, E1   -41.616, E3 +364336.851}
SPL {X  -157.709, Y  +713.973, Z    +0.000, E1   -41.360, E3 +364350.634}
SPL {X  -156.530, Y  +718.319, Z    +0.000, E1   -41.164, E3 +364361.578}
SPL {X  -155.547, Y  +721.618, Z    +0.000, E1   -40.968, E3 +364370.202}
SPL {X  -151.388, Y  +733.433, Z    +0.000, E1   -44.269, E3 +364377.905}
SPL {X  -144.352, Y  +748.818, Z    +0.000, E1   -40.701, E3 +364446.940}
SPL {X  -143.859, Y  +749.757, Z    +0.000, E1   -39.148, E3 +364474.888}
ENDSPLINE

SPLINE
SPL {X  -159.245, Y  +707.432, Z    +0.000, E1   -21.244, E3 +364506.921}
SPL {X  -162.277, Y  +686.791, Z    +0.000, E1   -10.607, E3 +364508.332}
SPL {X  -162.766, Y  +677.687, Z    +0.000, E1    -5.239, E3 +364510.521}
SPL {X  -162.820, Y  +671.059, Z    +0.000, E1    -0.934, E3 +364510.877}
SPL {X  -162.820, Y  +665.599, Z    +0.000, E1    +3.424, E3 +364511.327}
SPL {X  -162.820, Y  +661.024, Z    +0.000, E1    +7.880, E3 +364510.796}
SPL {X  -162.820, Y  +654.280, Z    +0.000, E1   +14.617, E3 +364511.513}
SPL {X  -162.820, Y  +638.947, Z    +0.000, E1   +31.033, E3 +364509.566}
SPL {X  -162.820, Y  +608.150, Z    +0.000, E1   +43.921, E3 +364535.799}
SPL {X  -162.820, Y  +574.255, Z    +0.000, E1   +46.562, E3 +364585.593}
ENDSPLINE

SPLINE
SPL {X  -162.820, Y  +579.440, Z    +0.000, E1   +42.450, E3 +364598.781}
ENDSPLINE

SPLINE
SPL {X  -162.820, Y  +574.443, Z    +0.000, E1   +42.333, E3 +364610.876}
SPL {X  -162.820, Y  +568.554, Z    +0.000, E1   +42.362, E3 +364624.238}
SPL {X  -162.820, Y  +561.474, Z    +0.000, E1   +42.369, E3 +364640.423}
SPL {X  -162.820, Y  +554.421, Z    +0.000, E1   +42.414, E3 +364656.247}
SPL {X  -162.820, Y  +547.774, Z    +0.000, E1   +42.344, E3 +364671.821}
SPL {X  -162.820, Y  +541.056, Z    +0.000, E1   +42.452, E3 +364686.482}
SPL {X  -162.820, Y  +535.223, Z    +0.000, E1   +42.386, E3 +364700.176}
SPL {X  -162.820, Y  +529.084, Z    +0.000, E1   +42.400, E3 +364714.099}
SPL {X  -162.820, Y  +524.911, Z    +0.000, E1   +42.325, E3 +364723.945}
SPL {X  -162.820, Y  +519.984, Z    +0.000, E1   +42.385, E3 +364735.015}
SPL {X  -162.820, Y  +512.536, Z    +0.000, E1   +42.385, E3 +364752.126}
SPL {X  -162.820, Y  +505.746, Z    +0.000, E1   +42.400, E3 +364767.370}
SPL {X  -162.820, Y  +500.461, Z    +0.000, E1   +42.387, E3 +364779.498}
SPL {X  -162.820, Y  +494.841, Z    +0.000, E1   +42.316, E3 +364792.824}
SPL {X  -162.820, Y  +486.958, Z    +0.000, E1   +42.460, E3 +364810.117}
SPL {X  -162.820, Y  +466.305, Z    +0.000, E1   +47.564, E3 +364823.124}
SPL {X  -162.820, Y  +462.532, Z    +0.000, E1   +47.610, E3 +364830.008}
SPL {X  -162.820, Y  +458.830, Z    +0.000, E1   +46.994, E3 +364841.008}
SPL {X  -162.820, Y  +455.537, Z    +0.000, E1   +45.900, E3 +364853.827}
SPL {X  -162.820, Y  +451.000, Z    +0.000, E1   +45.084, E3 +364868.202}
SPL {X  -162.820, Y  +442.850, Z    +0.000, E1   +44.856, E3 +364886.579}
SPL {X  -162.820, Y  +435.902, Z    +0.000, E1   +44.853, E3 +364900.944}
SPL {X  -162.820, Y  +429.336, Z    +0.000, E1   +44.917, E3 +364914.462}
SPL {X  -162.820, Y  +423.193, Z    +0.000, E1   +44.819, E3 +364927.721}
SPL {X  -162.820, Y  +416.810, Z    +0.000, E1   +44.932, E3 +364940.609}
SPL {X  -162.820, Y  +408.782, Z    +0.000, E1   +44.820, E3 +364958.040}
SPL {X  -162.820, Y  +401.619, Z    +0.000, E1   +44.978, E3 +364971.961}
SPL {X  -162.820, Y  +394.771, Z    +0.000, E1   +44.856, E3 +364987.201}
SPL {X  -162.820, Y  +387.883, Z    +0.000, E1   +44.837, E3 +365001.554}
SPL {X  -162.820, Y  +382.755, Z    +0.000, E1   +44.828, E3 +365012.347}
SPL {X  -162.796, Y  +377.700, Z    +0.000, E1   +44.829, E3 +365022.928}
SPL {X  -162.619, Y  +372.412, Z    +0.000, E1   +44.928, E3 +365033.387}
SPL {X  -162.311, Y  +367.633, Z    +0.000, E1   +44.798, E3 +365044.154}
SPL {X  -161.766, Y  +362.002, Z    +0.000, E1   +44.644, E3 +365056.913}
SPL {X  -161.043, Y  +356.508, Z    +0.000, E1   +44.528, E3 +365069.027}
SPL {X  -160.417, Y  +352.631, Z    +0.000, E1   +44.411, E3 +365077.758}
SPL {X  -159.536, Y  +347.962, Z    +0.000, E1   +44.302, E3 +365088.285}
SPL {X  -158.195, Y  +341.969, Z    +0.000, E1   +44.082, E3 +365102.067}
SPL {X  -156.950, Y  +337.174, Z    +0.000, E1   +43.768, E3 +365113.758}
SPL {X  -155.654, Y  +332.729, Z    +0.000, E1   +43.534, E3 +365124.400}
SPL {X  -153.067, Y  +324.996, Z    +0.000, E1   +44.257, E3 +365136.454}
SPL {X  -147.786, Y  +312.164, Z    +0.000, E1   +47.292, E3 +365145.185}
SPL {X  -142.680, Y  +302.060, Z    +0.000, E1   +42.084, E3 +365208.557}
ENDSPLINE

SPLINE
SPL {X  -151.184, Y  +320.053, Z    +0.000, E1   +32.435, E3 +365275.800}
SPL {X  -158.917, Y  +345.064, Z    +0.000, E1   +21.858, E3 +365277.148}
SPL {X  -161.350, Y  +358.672, Z    +0.000, E1   +15.089, E3 +365279.851}
SPL {X  -162.491, Y  +370.147, Z    +0.000, E1    +8.815, E3 +365282.786}
SPL {X  -162.771, Y  +376.522, Z    +0.000, E1    +5.005, E3 +365282.395}
SPL {X  -162.820, Y  +381.116, Z    +0.000, E1    +2.017, E3 +365282.729}
SPL {X  -162.820, Y  +384.427, Z    +0.000, E1    -0.390, E3 +365283.133}
SPL {X  -162.820, Y  +387.736, Z    +0.000, E1    -3.142, E3 +365282.413}
SPL {X  -162.820, Y  +391.456, Z    +0.000, E1    -6.603, E3 +365283.200}
SPL {X  -162.820, Y  +397.032, Z    +0.000, E1   -12.435, E3 +365282.647}
SPL {X  -162.820, Y  +406.111, Z    +0.000, E1   -22.010, E3 +365283.699}
SPL {X  -162.820, Y  +418.653, Z    +0.000, E1   -36.657, E3 +365278.051}
SPL {X  -162.820, Y  +440.590, Z    +0.000, E1   -50.152, E3 +365283.297}
SPL {X  -162.820, Y  +447.889, Z    +0.000, E1   -43.424, E3 +365314.443}
SPL {X  -162.820, Y  +479.020, Z    +0.000, E1   -47.189, E3 +365354.019}
ENDSPLINE

SPLINE
SPL {X  -162.820, Y  +474.886, Z    +0.000, E1   -43.721, E3 +365365.903}
ENDSPLINE

SPLINE
SPL {X  -162.820, Y  +476.137, Z    +0.000, E1   -42.304, E3 +365377.017}
SPL {X  -162.820, Y  +480.895, Z    +0.000, E1   -42.223, E3 +365388.476}
SPL {X  -162.820, Y  +485.782, Z    +0.000, E1   -42.348, E3 +365398.821}
SPL {X  -162.820, Y  +489.480, Z    +0.000, E1   -42.230, E3 +365408.048}
SPL {X  -162.820, Y  +494.825, Z    +0.000, E1   -42.287, E3 +365419.996}
SPL {X  -162.820, Y  +501.909, Z    +0.000, E1   -42.324, E3 +365436.182}
SPL {X  -162.820, Y  +508.157, Z    +0.000, E1   -42.280, E3 +365450.513}
SPL {X  -162.820, Y  +513.215, Z    +0.000, E1   -42.304, E3 +365462.043}
SPL {X  -162.820, Y  +520.311, Z    +0.000, E1   -42.317, E3 +365478.341}
SPL {X  -162.820, Y  +526.529, Z    +0.000, E1   -42.247, E3 +365492.811}
SPL {X  -162.820, Y  +531.715, Z    +0.000, E1   -42.312, E3 +365504.333}
SPL {X  -162.820, Y  +537.459, Z    +0.000, E1   -42.308, E3 +365517.592}
SPL {X  -162.820, Y  +542.643, Z    +0.000, E1   -42.173, E3 +365530.184}
SPL {X  -162.820, Y  +549.160, Z    +0.000, E1   -42.387, E3 +365543.943}
SPL {X  -162.820, Y  +554.884, Z    +0.000, E1   -42.207, E3 +365558.028}
SPL {X  -162.820, Y  +561.114, Z    +0.000, E1   -42.336, E3 +365571.608}
SPL {X  -162.820, Y  +566.097, Z    +0.000, E1   -42.118, E3 +365584.219}
SPL {X  -162.820, Y  +571.654, Z    +0.000, E1   -42.313, E3 +365595.872}
SPL {X  -162.820, Y  +577.246, Z    +0.000, E1   -42.284, E3 +365608.837}
SPL {X  -162.820, Y  +582.233, Z    +0.000, E1   -42.188, E3 +365620.817}
SPL {X  -162.820, Y  +588.138, Z    +0.000, E1   -42.308, E3 +365633.715}
SPL {X  -162.820, Y  +593.999, Z    +0.000, E1   -42.301, E3 +365647.125}
SPL {X  -162.820, Y  +599.194, Z    +0.000, E1   -42.235, E3 +365659.430}
SPL {X  -162.820, Y  +604.595, Z    +0.000, E1   -42.290, E3 +365671.461}
SPL {X  -162.820, Y  +609.630, Z    +0.000, E1   -42.276, E3 +365683.087}
SPL {X  -162.820, Y  +614.392, Z    +0.000, E1   -42.242, E3 +365694.187}
SPL {X  -162.820, Y  +620.424, Z    +0.000, E1   -42.277, E3 +365707.935}
SPL {X  -162.820, Y  +626.430, Z    +0.000, E1   -42.291, E3 +365721.485}
SPL {X  -162.820, Y  +631.865, Z    +0.000, E1   -42.327, E3 +365733.778}
SPL {X  -162.820, Y  +637.189, Z    +0.000, E1   -42.236, E3 +365746.452}
SPL {X  -162.820, Y  +642.066, Z    +0.000, E1   -42.247, E3 +365757.574}
SPL {X  -162.820, Y  +646.907, Z    +0.000, E1   -42.249, E3 +365768.693}
SPL {X  -162.820, Y  +652.374, Z    +0.000, E1   -42.262, E3 +365781.132}
SPL {X  -162.820, Y  +657.439, Z    +0.000, E1   -42.251, E3 +365792.805}
SPL {X  -162.820, Y  +663.328, Z    +0.000, E1   -42.283, E3 +365806.207}
SPL {X  -162.820, Y  +669.078, Z    +0.000, E1   -42.263, E3 +365819.403}
SPL {X  -162.819, Y  +673.910, Z    +0.000, E1   -42.244, E3 +365830.597}
SPL {X  -162.729, Y  +678.944, Z    +0.000, E1   -42.273, E3 +365841.965}
SPL {X  -162.479, Y  +684.035, Z    +0.000, E1   -42.168, E3 +365854.302}
SPL {X  -162.026, Y  +689.560, Z    +0.000, E1   -42.192, E3 +365866.791}
SPL {X  -161.446, Y  +694.609, Z    +0.000, E1   -42.094, E3 +365878.923}
SPL {X  -160.681, Y  +699.806, Z    +0.000, E1   -41.866, E3 +365892.206}
SPL {X  -159.658, Y  +705.434, Z    +0.000, E1   -41.735, E3 +365905.836}
SPL {X  -158.502, Y  +710.748, Z    +0.000, E1   -41.532, E3 +365919.183}
SPL {X  -157.452, Y  +714.962, Z    +0.000, E1   -41.276, E3 +365930.178}
SPL {X  -156.530, Y  +718.319, Z    +0.000, E1   -41.164, E3 +365938.501}
SPL {X  -155.547, Y  +721.618, Z    +0.000, E1   -40.968, E3 +365947.125}
SPL {X  -151.388, Y  +733.433, Z    +0.000, E1   -44.269, E3 +365954.828}
SPL {X  -144.352, Y  +748.818, Z    +0.000, E1   -40.701, E3 +366023.863}
SPL {X  -143.859, Y  +749.757, Z    +0.000, E1   -39.148, E3 +366051.811}
ENDSPLINE

SPLINE
SPL {X  -159.245, Y  +707.432, Z    +0.000, E1   -21.244, E3 +366083.844}
SPL {X  -162.277, Y  +686.791, Z    +0.000, E1   -10.607, E3 +366085.255}
SPL {X  -162.766, Y  +677.687, Z    +0.000, E1    -5.239, E3 +366087.444}
SPL {X  -162.820, Y  +671.059, Z    +0.000, E1    -0.934, E3 +366087.800}
SPL {X  -162.820, Y  +665.599, Z    +0.000, E1    +3.424, E3 +366088.250}
SPL {X  -162.820, Y  +661.024, Z    +0.000, E1    +7.880, E3 +366087.719}
SPL {X  -162.820, Y  +656.051, Z    +0.000, E1   +12.848, E3 +366088.586}
SPL {X  -162.820, Y  +650.794, Z    +0.000, E1   +18.580, E3 +366088.142}
SPL {X  -162.820, Y  +638.947, Z    +0.000, E1   +31.033, E3 +366086.490}
SPL {X  -162.820, Y  +608.150, Z    +0.000, E1   +43.921, E3 +366112.722}
SPL {X  -162.820, Y  +574.255, Z    +0.000, E1   +46.562, E3 +366162.516}
ENDSPLINE

SPLINE
SPL {X  -162.820, Y  +579.440, Z    +0.000, E1   +42.450, E3 +366175.704}
ENDSPLINE

